# B&R Automation Studio project EFI (part 10)

#### AssignDataComms.st
```iecst
ACTION AssignDataComms:

	//Active modbus slave diagnosis when module ok (cable plugged). To set to false just unplug de cable
	IF PowerMeter.Status.Comms.xModuleOk THEN
		PowerMeter.Parameters.xActiveSlaveDiagnosis := TRUE; //1: Diagnosis enabled; 0=Reset diagnosis historic
	END_IF

	////////////////
	//Read Registers

	//Current
	IF PowerMeter.Status.Comms.xModuleOk THEN
		PowerMeter.Inputs.Comms.EffectiveCurrentPhaseA := PowerMeter.Inputs.Comms.ReceivedDataModPowerMeter[16];
		PowerMeter.Inputs.Comms.EffectiveCurrentPhaseB := PowerMeter.Inputs.Comms.ReceivedDataModPowerMeter[17];
		PowerMeter.Inputs.Comms.EffectiveCurrentPhaseC := PowerMeter.Inputs.Comms.ReceivedDataModPowerMeter[18];
		PowerMeter.Inputs.Comms.EffectiveCurrentNeutral := PowerMeter.Inputs.Comms.ReceivedDataModPowerMeter[19];
		PowerMeter.Inputs.Comms.MaxCurrentAllPhases := PowerMeter.Inputs.Comms.ReceivedDataModPowerMeter[20];
		PowerMeter.Inputs.Comms.IgEarthDefectiveCurrent := PowerMeter.Inputs.Comms.ReceivedDataModPowerMeter[21];
		PowerMeter.Inputs.Comms.CurrentDifferential := PowerMeter.Inputs.Comms.ReceivedDataModPowerMeter[22];
		PowerMeter.Inputs.Comms.MaxEffectiveCurrentPhaseA := PowerMeter.Inputs.Comms.ReceivedDataModPowerMeter[23];
		PowerMeter.Inputs.Comms.MaxEffectiveCurrentPhaseB := PowerMeter.Inputs.Comms.ReceivedDataModPowerMeter[24];
		PowerMeter.Inputs.Comms.MaxEffectiveCurrentPhaseC := PowerMeter.Inputs.Comms.ReceivedDataModPowerMeter[25];
		PowerMeter.Inputs.Comms.MaxEffectiveCurrentNeutral := PowerMeter.Inputs.Comms.ReceivedDataModPowerMeter[26];

		//Frequency
		PowerMeter.Inputs.Comms.MaxIgEarthDefectiveCurrent := PowerMeter.Inputs.Comms.ReceivedDataModPowerMeter[28];
		PowerMeter.Inputs.Comms.MaxCurrentDifferential := PowerMeter.Inputs.Comms.ReceivedDataModPowerMeter[29];

		//Voltage
		PowerMeter.Inputs.Comms.EffectiveVoltagePhasesAB := PowerMeter.Inputs.Comms.ReceivedDataModPowerMeter[30];
		PowerMeter.Inputs.Comms.EffectiveVoltagePhasesBC := PowerMeter.Inputs.Comms.ReceivedDataModPowerMeter[31];
		PowerMeter.Inputs.Comms.EffectiveVoltagePhasesCA := PowerMeter.Inputs.Comms.ReceivedDataModPowerMeter[32];
		PowerMeter.Inputs.Comms.EffectiveVoltagePhasesAN := PowerMeter.Inputs.Comms.ReceivedDataModPowerMeter[33];
		PowerMeter.Inputs.Comms.EffectiveVoltagePhasesBN := PowerMeter.Inputs.Comms.ReceivedDataModPowerMeter[34];
		PowerMeter.Inputs.Comms.EffectiveVoltagePhasesCN := PowerMeter.Inputs.Comms.ReceivedDataModPowerMeter[35];
		PowerMeter.Inputs.Comms.Frequency := PowerMeter.Inputs.Comms.ReceivedDataModPowerMeter[36]/10;
		PowerMeter.Inputs.Comms.FrequencyMax := PowerMeter.Inputs.Comms.ReceivedDataModPowerMeter[37]/10;

		//Power
		PowerMeter.Inputs.Comms.ActivePowerPhaseA := PowerMeter.Inputs.Comms.ReceivedDataModPowerMeter[38];
		PowerMeter.Inputs.Comms.ActivePowerPhaseB := PowerMeter.Inputs.Comms.ReceivedDataModPowerMeter[39];
		PowerMeter.Inputs.Comms.ActivePowerPhaseC := PowerMeter.Inputs.Comms.ReceivedDataModPowerMeter[40];
		PowerMeter.Inputs.Comms.TotalActivePower := PowerMeter.Inputs.Comms.ReceivedDataModPowerMeter[41];
		PowerMeter.Inputs.Comms.ApparentPowerPhaseA := PowerMeter.Inputs.Comms.ReceivedDataModPowerMeter[42];
		PowerMeter.Inputs.Comms.ApparentPowerPhaseB := PowerMeter.Inputs.Comms.ReceivedDataModPowerMeter[43];
		PowerMeter.Inputs.Comms.ApparentPowerPhaseC := PowerMeter.Inputs.Comms.ReceivedDataModPowerMeter[44];
		PowerMeter.Inputs.Comms.TotalApparentPower := PowerMeter.Inputs.Comms.ReceivedDataModPowerMeter[45];
		PowerMeter.Inputs.Comms.ReactivePowerPhaseA := PowerMeter.Inputs.Comms.ReceivedDataModPowerMeter[46];
		PowerMeter.Inputs.Comms.ReactivePowerPhaseB := PowerMeter.Inputs.Comms.ReceivedDataModPowerMeter[47];
		PowerMeter.Inputs.Comms.ReactivePowerPhaseC := PowerMeter.Inputs.Comms.ReceivedDataModPowerMeter[48];
		PowerMeter.Inputs.Comms.TotalReactivePower := PowerMeter.Inputs.Comms.ReceivedDataModPowerMeter[49];

		//Total Harmonic Distortion) (THD)
		PowerMeter.Inputs.Comms.THDVoltageAB := PowerMeter.Inputs.Comms.ReceivedDataModPowerMeter[104];
		PowerMeter.Inputs.Comms.THDVoltageBC := PowerMeter.Inputs.Comms.ReceivedDataModPowerMeter[105];
		PowerMeter.Inputs.Comms.THDVoltageCA := PowerMeter.Inputs.Comms.ReceivedDataModPowerMeter[106];
		PowerMeter.Inputs.Comms.THDVoltageAN := PowerMeter.Inputs.Comms.ReceivedDataModPowerMeter[107];
		PowerMeter.Inputs.Comms.THDVoltageBN := PowerMeter.Inputs.Comms.ReceivedDataModPowerMeter[108];
		PowerMeter.Inputs.Comms.THDVoltageCN := PowerMeter.Inputs.Comms.ReceivedDataModPowerMeter[109];
		PowerMeter.Inputs.Comms.THDCurrentA := PowerMeter.Inputs.Comms.ReceivedDataModPowerMeter[110];
		PowerMeter.Inputs.Comms.THDCurrentB := PowerMeter.Inputs.Comms.ReceivedDataModPowerMeter[111];
		PowerMeter.Inputs.Comms.THDCurrentC := PowerMeter.Inputs.Comms.ReceivedDataModPowerMeter[112];
		PowerMeter.Inputs.Comms.TotalTHDCurrent := PowerMeter.Inputs.Comms.ReceivedDataModPowerMeter[113];
	END_IF

END_ACTION
```

### Program Logical/ExtPack/_Extras/SafetyControllerCtrl/SafetyControllerCtrl_v1/SafetyControllerCtrl (IEC)

#### AssignDataComms.st
```iecst
ACTION AssignDataComms:

	//Active modbus slave diagnosis when module ok (cable plugged). To set to false just unplug de cable
	IF SafetyController.Status.Comms.xModuleOk THEN
		SafetyController.Parameters.xActiveSlaveDiagnosis := TRUE; //1: Diagnosis enabled; 0=Reset diagnosis historic
	END_IF

	//Pre bits treatment

	//Write Registers

	//Read Registers
	IF SafetyController.Status.Comms.xModuleOk THEN

		SafetyController.Inputs.Comms.FieldbusProbeStatus := DataFromSafety[11];

		IF NOT SafetyController.Parameters.xSimulationMode THEN
			//Software version
			SafetyController.Status.Version.0 := SafetyController.Inputs.Comms.FieldbusProbeStatus.0;
			SafetyController.Status.Version.1 := SafetyController.Inputs.Comms.FieldbusProbeStatus.1;
			SafetyController.Status.Version.2 := SafetyController.Inputs.Comms.FieldbusProbeStatus.2;
		END_IF

		CASE gMachine.Pt.ConfigNameID OF
			GC_CONFIG_1BK8BAR_NOZ2_ID:
				CASE SafetyController.Status.Version OF
					1: SafetyController.Status.Type := SAFETYCONTROLLERTY_DEFAULT;
					2: SafetyController.Status.Type := SAFETYCONTROLLERTY_DEFAULT;
					3: SafetyController.Status.Type := SAFETYCONTROLLERTY_CUBE_ALPHA;
					4: SafetyController.Status.Type := SAFETYCONTROLLERTY_SD;

					ELSE SafetyController.Status.Type := SAFETYCONTROLLERTY_UNDEFINED;
				END_CASE

			GC_CONFIG_1BK8BAR_NOZ2_AQ_ID:
				CASE SafetyController.Status.Version OF
					1: SafetyController.Status.Type := SAFETYCONTROLLERTY_NOZ2_AQ;

					ELSE SafetyController.Status.Type := SAFETYCONTROLLERTY_UNDEFINED;
				END_CASE

			GC_CONFIG_1BK7BAR_CUBE_ID:
				//To uncomment this code when first release that supports CUBE will be launched. So we will be sure safety controller version matches properly
				CASE SafetyController.Status.Version OF
					1: SafetyController.Status.Type := SAFETYCONTROLLERTY_CUBE;

					ELSE SafetyController.Status.Type := SAFETYCONTROLLERTY_UNDEFINED;
				END_CASE

			GC_CONFIG_1BK10BAR_MECANO_ID:
				//To uncomment this code when first release that supports CUBE will be launched. So we will be sure safety controller version matches properly
				CASE SafetyController.Status.Version OF
					1: SafetyController.Status.Type := SAFETYCONTROLLERTY_MECANO;

					ELSE SafetyController.Status.Type := SAFETYCONTROLLERTY_UNDEFINED;
				END_CASE

			GC_CONFIG_SIMTEST_ID:
				CASE gMachine.Pt.MachineModel OF
					Type_NOZ_2_AQ:
						SafetyController.Status.Type := SAFETYCONTROLLERTY_NOZ2_AQ;

					Type_NOZ_2_UV,
					Type_NOZ_2_UV_White:
						SafetyController.Status.Type := SAFETYCONTROLLERTY_DEFAULT;

					Type_CUBE,
					Type_CUBE_INSPECTION,
					Type_CUBE_GULLIVER,
					Type_CUBE_GULLIVER_INSPECTION:
						SafetyController.Status.Type := SAFETYCONTROLLERTY_CUBE;

					Type_MECANO_UV_WHITE,
					Type_MECANO_UV_OPV,
					Type_MECANO_UV_WHITE_OPV:
						SafetyController.Status.Type := SAFETYCONTROLLERTY_MECANO;

					ELSE SafetyController.Status.Type := SAFETYCONTROLLERTY_UNDEFINED;
				END_CASE

		END_CASE

		IF NOT SafetyController.Parameters.xSimulationMode THEN
			CASE SafetyController.Status.Type OF
				//Cube machine
				SAFETYCONTROLLERTY_CUBE:
					SafetyController.Inputs.Comms.SystemStatus := UINT_TO_USINT(DataFromSafety[0] AND 16#00FF);
					SafetyController.Inputs.Comms.ExpansionModule[0] := UINT_TO_USINT(DataFromSafety[1] AND 16#00FF); 			// CP0802
					SafetyController.Inputs.Comms.ExpansionModule[1] := UINT_TO_USINT(SHR((DataFromSafety[1] AND 16#FF00),8)); 	//DI16-0
					SafetyController.Inputs.Comms.ExpansionModule[2] := UINT_TO_USINT(DataFromSafety[2] AND 16#00FF);			//R04-0

					//Fieldbus probe
					//Inputs
					SafetyController.Inputs.xPrinterRearDoorSwitch := SafetyController.Inputs.Comms.FieldbusProbeStatus.3;
					SafetyController.Inputs.xPrinterMaintenanceKey := SafetyController.Inputs.Comms.FieldbusProbeStatus.4;
					SafetyController.Inputs.xHmiSwitch := SafetyController.Inputs.Comms.FieldbusProbeStatus.5;
					SafetyController.Inputs.xPrinterFrontDoorSwitch := SafetyController.Inputs.Comms.FieldbusProbeStatus.6;
					SafetyController.Inputs.xPrinterBacksideEstop := SafetyController.Inputs.Comms.FieldbusProbeStatus.7;
					SafetyController.Inputs.xPrinterFrontsideEstop := SafetyController.Inputs.Comms.FieldbusProbeStatus.8;
					SafetyController.Inputs.xX5Consent := SafetyController.Inputs.Comms.FieldbusProbeStatus.9;
					SafetyController.Inputs.xFanDoorSwitch := SafetyController.Inputs.Comms.FieldbusProbeStatus.12;

					//Outputs
					SafetyController.Outputs.xEnablePrinter1 := SafetyController.Inputs.Comms.FieldbusProbeStatus.11; //Revisar por qué esta asignación no funciona bien
					SafetyController.Outputs.xPrinterToX5 := SafetyController.Inputs.Comms.FieldbusProbeStatus.11;

				SAFETYCONTROLLERTY_DEFAULT,
				SAFETYCONTROLLERTY_CUBE_ALPHA,
				SAFETYCONTROLLERTY_SD:
					SafetyController.Inputs.Comms.SystemStatus := UINT_TO_USINT(DataFromSafety[0] AND 16#00FF);
					SafetyController.Inputs.Comms.ExpansionModule[0] := UINT_TO_USINT(DataFromSafety[1] AND 16#00FF);			// CP0802
					SafetyController.Inputs.Comms.ExpansionModule[1] := UINT_TO_USINT(SHR((DataFromSafety[1] AND 16#FF00),8));	//MX0802
					SafetyController.Inputs.Comms.ExpansionModule[2] := UINT_TO_USINT(DataFromSafety[2] AND 16#00FF);			//DI16-0
					SafetyController.Inputs.Comms.ExpansionModule[3] := UINT_TO_USINT(SHR((DataFromSafety[2] AND 16#FF00),8));	//DI16-1
					SafetyController.Inputs.Comms.ExpansionModule[4] := UINT_TO_USINT(DataFromSafety[3] AND 16#00FF);			//R04-0
					SafetyController.Inputs.Comms.ExpansionModule[5] := UINT_TO_USINT(SHR((DataFromSafety[3] AND 16#FF00),8));	//R04-1
					SafetyController.Inputs.Comms.ExpansionModule[6] := UINT_TO_USINT(DataFromSafety[4] AND 16#00FF);			//R04-2

					//SafetyController.Inputs.Comms.FieldbusProbeStatus := DataFromSafety[11];
					SafetyController.Inputs.Comms.OSSDStatus := DataFromSafety[13];
					SafetyController.Inputs.Comms.DiagnosticCode := DataFromSafety[14];

					//Post bit treatment
					//Fieldbus: Currently there is no need to acknowledge fiedlbus inputs set in SoSafe program so info coming from inputs is enough

					//Modules physical inputs
					//Ancillaries
					SafetyController.Inputs.xFeederEstop			:= SafetyController.Inputs.Comms.FieldbusProbeStatus.8; //SafetyController.Inputs.Comms.ExpansionModule[1].0;
					SafetyController.Inputs.xPrimerEstop 			:= SafetyController.Inputs.Comms.FieldbusProbeStatus.9; //SafetyController.Inputs.Comms.ExpansionModule[1].2;
					SafetyController.Inputs.xOvervarnishEstop 		:= SafetyController.Inputs.Comms.FieldbusProbeStatus.14; //SafetyController.Inputs.Comms.ExpansionModule[2].4;
					SafetyController.Inputs.xStackerEstop 			:= SafetyController.Inputs.Comms.FieldbusProbeStatus.15; //SafetyController.Inputs.Comms.ExpansionModule[2].0;
					SafetyController.Inputs.xSarmEstop				:= SafetyController.Inputs.Comms.FieldbusProbeStatus.7;

					//Dryer
					SafetyController.Inputs.xDryerBacksideEstop 	:= SafetyController.Inputs.Comms.FieldbusProbeStatus.12; //SafetyController.Inputs.Comms.ExpansionModule[1].4;
					SafetyController.Inputs.xDryerFrontsideEstop 	:= SafetyController.Inputs.Comms.FieldbusProbeStatus.13; //SafetyController.Inputs.Comms.ExpansionModule[1].6;
					SafetyController.Inputs.xDryerFrontDoorSwitch1	:= SafetyController.Inputs.Comms.FieldbusProbeStatus.3; //SafetyController.Inputs.Comms.ExpansionModule[2].6;
					SafetyController.Inputs.xDryerFrontDoorSwitch2	:= SafetyController.Inputs.Comms.FieldbusProbeStatus.4; //SafetyController.Inputs.Comms.ExpansionModule[3].4;
					SafetyController.Inputs.xDryerBackDoorSwitch1	:= SafetyController.Inputs.Comms.FieldbusProbeStatus.5; //SafetyController.Inputs.Comms.ExpansionModule[3].6;
					SafetyController.Inputs.xDryerBackDoorSwitch2	:= SafetyController.Inputs.Comms.FieldbusProbeStatus.6; //SafetyController.Inputs.Comms.ExpansionModule[4].0;
					SafetyController.Inputs.xDryerMaintenanceKey	:= SafetyController.Inputs.Comms.ExpansionModule[4].3;
					SafetyController.Inputs.xDryerBlowersEnable		:= SafetyController.Inputs.Comms.ExpansionModule[2].3;

					//Printer
					SafetyController.Inputs.xPrinterMaintenanceKey 	:= SafetyController.Inputs.Comms.ExpansionModule[4].2;
					SafetyController.Inputs.xPrinterBlowersEnable	:= SafetyController.Inputs.Comms.ExpansionModule[2].2;
					SafetyController.Inputs.xPrinterBlowersSwitch	:= TRUE; //SafetyController.Inputs.Comms.FieldbusProbeStatus.2;
					SafetyController.Inputs.xPrinterLightCurtain 	:= SafetyController.Inputs.Comms.ExpansionModule[0].0;
					SafetyController.Inputs.xPrinterDoorLock 		:= SafetyController.Inputs.Comms.ExpansionModule[0].2;
					SafetyController.Inputs.xPrinterBacksideEstop 	:= SafetyController.Inputs.Comms.FieldbusProbeStatus.10;
					SafetyController.Inputs.xPrinterFrontsideEstop 	:= SafetyController.Inputs.Comms.FieldbusProbeStatus.11;

					//OSSD Outputs
					SafetyController.Outputs.xEnablePrinter1 := SafetyController.Inputs.Comms.OSSDStatus.0;
					//SafetyController.Outputs.xEnablePrinter2 := SafetyController.Inputs.Comms.OSSDStatus.1;
					SafetyController.Outputs.xEnablePrinterBlowers1 := SafetyController.Inputs.Comms.OSSDStatus.1;
					//SafetyController.Outputs.xEnablePrinterBlowers2	:= SafetyController.Inputs.Comms.OSSDStatus.3;
					SafetyController.Outputs.xEnableDryer1	:= SafetyController.Inputs.Comms.OSSDStatus.2;
					//SafetyController.Outputs.xEnableDryer2	:= SafetyController.Inputs.Comms.OSSDStatus.5;

				SAFETYCONTROLLERTY_MECANO:
					SafetyController.Inputs.Comms.SystemStatus := UINT_TO_USINT(DataFromSafety[0] AND 16#00FF);
					SafetyController.Inputs.Comms.ExpansionModule[0] := UINT_TO_USINT(DataFromSafety[1] AND 16#00FF);			// CP0802
					SafetyController.Inputs.Comms.ExpansionModule[1] := UINT_TO_USINT(SHR((DataFromSafety[1] AND 16#FF00),8));	//MX0802
					SafetyController.Inputs.Comms.ExpansionModule[2] := UINT_TO_USINT(DataFromSafety[2] AND 16#00FF);			//DI16-0
					SafetyController.Inputs.Comms.ExpansionModule[3] := UINT_TO_USINT(SHR((DataFromSafety[2] AND 16#FF00),8));	//DI16-1
					SafetyController.Inputs.Comms.ExpansionModule[4] := UINT_TO_USINT(DataFromSafety[3] AND 16#00FF);			//R04-0
					SafetyController.Inputs.Comms.ExpansionModule[5] := UINT_TO_USINT(SHR((DataFromSafety[3] AND 16#FF00),8));	//R04-1
					SafetyController.Inputs.Comms.ExpansionModule[6] := UINT_TO_USINT(DataFromSafety[4] AND 16#00FF);			//R04-2

					//SafetyController.Inputs.Comms.FieldbusProbeStatus := DataFromSafety[11];
					SafetyController.Inputs.Comms.OSSDStatus := DataFromSafety[13];
					SafetyController.Inputs.Comms.DiagnosticCode := DataFromSafety[14];

					//Post bit treatment
					//Modules physical inputs
					//Ancillaries
					SafetyController.Inputs.xFeederEstop			:= SafetyController.Inputs.Comms.FieldbusProbeStatus.8;
					SafetyController.Inputs.xPrimerEstop 			:= SafetyController.Inputs.Comms.FieldbusProbeStatus.9;
					SafetyController.Inputs.xOvervarnishEstop 		:= SafetyController.Inputs.Comms.FieldbusProbeStatus.14;
					SafetyController.Inputs.xStackerEstop 			:= SafetyController.Inputs.Comms.FieldbusProbeStatus.15;
					SafetyController.Inputs.xSarmEstop				:= SafetyController.Inputs.Comms.FieldbusProbeStatus.7;

					//Printer
					SafetyController.Inputs.xPrinterMaintenanceKey 	:= SafetyController.Inputs.Comms.FieldbusProbeStatus.5;
					SafetyController.Inputs.xPrinterBlowersEnable	:= SafetyController.Inputs.Comms.ExpansionModule[2].2;
					SafetyController.Inputs.xPrinterBlowersSwitch	:= SafetyController.Inputs.Comms.FieldbusProbeStatus.6;
					SafetyController.Inputs.xPrinterLightCurtain 	:= SafetyController.Inputs.Comms.FieldbusProbeStatus.3;
					SafetyController.Inputs.xPrinterDoorLock 		:= SafetyController.Inputs.Comms.FieldbusProbeStatus.4;
					SafetyController.Inputs.xPrinterBacksideEstop 	:= SafetyController.Inputs.Comms.FieldbusProbeStatus.10;
					SafetyController.Inputs.xPrinterFrontsideEstop 	:= SafetyController.Inputs.Comms.FieldbusProbeStatus.11;

					//OSSD Outputs
					SafetyController.Outputs.xEnablePrinter1 		:= SafetyController.Inputs.Comms.OSSDStatus.0;
					SafetyController.Outputs.xEnablePrinterBlowers1 := SafetyController.Inputs.Comms.OSSDStatus.1;

				SAFETYCONTROLLERTY_NOZ2_AQ:
					SafetyController.Inputs.Comms.SystemStatus := UINT_TO_USINT(DataFromSafety[0] AND 16#00FF);
					SafetyController.Inputs.Comms.ExpansionModule[0] := UINT_TO_USINT(DataFromSafety[1] AND 16#00FF);			// CP0802
					SafetyController.Inputs.Comms.ExpansionModule[1] := UINT_TO_USINT(SHR((DataFromSafety[1] AND 16#FF00),8));	//MX0802
					SafetyController.Inputs.Comms.ExpansionModule[2] := UINT_TO_USINT(DataFromSafety[2] AND 16#00FF);			//DI16-0
					SafetyController.Inputs.Comms.ExpansionModule[3] := UINT_TO_USINT(SHR((DataFromSafety[2] AND 16#FF00),8));	//DI16-1
					SafetyController.Inputs.Comms.ExpansionModule[4] := UINT_TO_USINT(DataFromSafety[3] AND 16#00FF);			//R04-0
					SafetyController.Inputs.Comms.ExpansionModule[5] := UINT_TO_USINT(SHR((DataFromSafety[3] AND 16#FF00),8));	//R04-1
					SafetyController.Inputs.Comms.ExpansionModule[6] := UINT_TO_USINT(DataFromSafety[4] AND 16#00FF);			//R04-2

					SafetyController.Inputs.Comms.OSSDStatus := DataFromSafety[13];
					SafetyController.Inputs.Comms.DiagnosticCode := DataFromSafety[14];

					//Post bit treatment
					//Fieldbus: Currently there is no need to acknowledge fiedlbus inputs set in SoSafe program so info coming from inputs is enough

					//Modules physical inputs
					//Ancillaries
					SafetyController.Inputs.xFeederEstop			:= SafetyController.Inputs.Comms.FieldbusProbeStatus.8; //SafetyController.Inputs.Comms.ExpansionModule[1].0;
					SafetyController.Inputs.xPrimerEstop 			:= SafetyController.Inputs.Comms.FieldbusProbeStatus.9; //SafetyController.Inputs.Comms.ExpansionModule[1].2;
					SafetyController.Inputs.xOvervarnishEstop 		:= SafetyController.Inputs.Comms.FieldbusProbeStatus.14; //SafetyController.Inputs.Comms.ExpansionModule[2].4;
					SafetyController.Inputs.xStackerEstop 			:= SafetyController.Inputs.Comms.FieldbusProbeStatus.15; //SafetyController.Inputs.Comms.ExpansionModule[2].0;

					//Dryer
					SafetyController.Inputs.xDryerBacksideEstop 	:= SafetyController.Inputs.Comms.FieldbusProbeStatus.12; //SafetyController.Inputs.Comms.ExpansionModule[1].4;
					SafetyController.Inputs.xDryerFrontsideEstop 	:= SafetyController.Inputs.Comms.FieldbusProbeStatus.13; //SafetyController.Inputs.Comms.ExpansionModule[1].6;
					SafetyController.Inputs.xDryerFrontDoorSwitch1	:= SafetyController.Inputs.Comms.FieldbusProbeStatus.3; //SafetyController.Inputs.Comms.ExpansionModule[2].6;
					SafetyController.Inputs.xDryerFrontDoorSwitch2	:= SafetyController.Inputs.Comms.FieldbusProbeStatus.4; //SafetyController.Inputs.Comms.ExpansionModule[3].4;
					SafetyController.Inputs.xDryerBackDoorSwitch1	:= SafetyController.Inputs.Comms.FieldbusProbeStatus.5; //SafetyController.Inputs.Comms.ExpansionModule[3].6;
					SafetyController.Inputs.xDryerBackDoorSwitch2	:= SafetyController.Inputs.Comms.FieldbusProbeStatus.6; //SafetyController.Inputs.Comms.ExpansionModule[4].0;
					SafetyController.Inputs.xDryerMaintenanceKey	:= SafetyController.Inputs.Comms.ExpansionModule[4].3;
					SafetyController.Inputs.xDryerBlowersEnable		:= SafetyController.Inputs.Comms.ExpansionModule[2].3;

					//Printer
					SafetyController.Inputs.xPrinterMaintenanceKey 	:= SafetyController.Inputs.Comms.ExpansionModule[4].2;
					SafetyController.Inputs.xPrinterBlowersEnable	:= SafetyController.Inputs.Comms.ExpansionModule[2].2;
					SafetyController.Inputs.xPrinterBlowersSwitch	:= TRUE;
					SafetyController.Inputs.xPrinterLightCurtain 	:= SafetyController.Inputs.Comms.ExpansionModule[0].0;
					SafetyController.Inputs.xPrinterDoorLock 		:= SafetyController.Inputs.Comms.ExpansionModule[0].2;
					SafetyController.Inputs.xPrinterBacksideEstop 	:= SafetyController.Inputs.Comms.FieldbusProbeStatus.10;
					SafetyController.Inputs.xPrinterFrontsideEstop 	:= SafetyController.Inputs.Comms.FieldbusProbeStatus.11;

					//OSSD Outputs
					SafetyController.Outputs.xEnablePrinter1 := SafetyController.Inputs.Comms.OSSDStatus.0;
					SafetyController.Outputs.xEnablePrinterBlowers1 := SafetyController.Inputs.Comms.OSSDStatus.1;
					SafetyController.Outputs.xEnableDryer1	:= SafetyController.Inputs.Comms.OSSDStatus.2;

				ELSE
					SafetyController.Inputs := ResetSafetyInputs;
					SafetyController.Outputs := ResetSafetyOutputs;

			END_CASE
		END_IF
	END_IF

END_ACTION
```

#### Alarms.st
```iecst
ACTION Alarms:

	//Reset Alarms with an external order to reset
	IF SafetyController.Commands.xReset THEN
		ResetAlarms;
	END_IF

	//Saving modbus slave status when comms error raises
	IF EDGEPOS (SafetyController.Alarms.xCommsError) THEN
		ModSlaveState := SafetyController.Status.Comms.ModSlaveState;
		LastError := SafetyController.Status.Comms.LastError;
		LastErrorBlockNum := SafetyController.Status.Comms.LastErrorBlockNum;
	END_IF

	//Alarms related to comms
	IF SafetyController.Status.Comms.xModuleOk THEN

		CASE SafetyController.Status.Type OF
			//Cube machine
			SAFETYCONTROLLERTY_CUBE:

				SafetyController.Alarms.xAlrPrinterRearDoorSwitch := NOT SafetyController.Inputs.xPrinterRearDoorSwitch AND NOT SafetyController.Inputs.xPrinterMaintenanceKey;
				SafetyController.Alarms.xAlrHmiSwitch := NOT SafetyController.Inputs.xHmiSwitch;
				SafetyController.Alarms.xAlrPrinterFrontDoorSwitch := NOT SafetyController.Inputs.xPrinterFrontDoorSwitch AND NOT SafetyController.Inputs.xPrinterMaintenanceKey;
				SafetyController.Alarms.xAlrPrinterFanDoorSwitch := NOT SafetyController.Inputs.xFanDoorSwitch;

				SafetyController.Alarms.xAlrPrinterEStops := 	NOT SafetyController.Inputs.xPrinterBacksideEstop OR
																NOT SafetyController.Inputs.xPrinterFrontsideEstop;

				SafetyController.Alarms.xAlrPrinter := 	SafetyController.Alarms.xAlrPrinterRearDoorSwitch OR
														SafetyController.Alarms.xAlrHmiSwitch OR
														SafetyController.Alarms.xAlrPrinterFrontDoorSwitch OR
														SafetyController.Alarms.xAlrPrinterFanDoorSwitch OR
														SafetyController.Alarms.xAlrPrinterEStops;

				SafetyController.Alarms.xAlrPrinterDoorLockKeyActivated := SafetyController.Inputs.xPrinterMaintenanceKey;

				SafetyController.Alarms.xAlrFeeder := NOT SafetyController.Inputs.xX5Consent;

				SafetyController.Alarms.xAlrPrinterFrontEstop :=  NOT SafetyController.Inputs.xPrinterFrontsideEstop;
				SafetyController.Alarms.xAlrPrinterRearEstop := NOT SafetyController.Inputs.xPrinterBacksideEstop;

			SAFETYCONTROLLERTY_DEFAULT,
			SAFETYCONTROLLERTY_CUBE_ALPHA,
			SAFETYCONTROLLERTY_SD,
			SAFETYCONTROLLERTY_MECANO:
				tonAlarmFeeder.IN := NOT SafetyController.Inputs.xFeederEstop;
				tonAlarmFeeder.PT := T#3s;
				tonAlarmFeeder();
				SafetyController.Alarms.xAlrFeeder := tonAlarmFeeder.Q;

				tonAlarmPrimer.IN := NOT SafetyController.Inputs.xPrimerEstop;
				tonAlarmPrimer.PT := T#3s;
				tonAlarmPrimer();
				SafetyController.Alarms.xAlrPrimer := tonAlarmPrimer.Q;

				SafetyController.Alarms.xAlrPrinter := 	NOT SafetyController.Inputs.xPrinterLightCurtain OR
														NOT SafetyController.Inputs.xPrinterDoorLock OR
														NOT SafetyController.Inputs.xPrinterBacksideEstop OR
														NOT SafetyController.Inputs.xPrinterFrontsideEstop;

				SafetyController.Alarms.xAlrPrinterEStops := 	NOT SafetyController.Inputs.xPrinterBacksideEstop OR
																NOT SafetyController.Inputs.xPrinterFrontsideEstop;

				tonAlarmOverVarnish.IN := NOT SafetyController.Inputs.xOvervarnishEstop;
				tonAlarmOverVarnish.PT := T#3s;
				tonAlarmOverVarnish();
				SafetyController.Alarms.xAlrOverVarnish := tonAlarmOverVarnish.Q;

				tonAlarmStacker.IN := NOT SafetyController.Inputs.xStackerEstop;
				tonAlarmStacker.PT := T#3s;
				tonAlarmStacker();
				SafetyController.Alarms.xAlrStacker := tonAlarmStacker.Q;

				IF SafetyController.Status.Type = SAFETYCONTROLLERTY_SD OR SafetyController.Status.Type = SAFETYCONTROLLERTY_MECANO THEN
					tonAlarmSarm.IN := NOT SafetyController.Inputs.xSarmEstop;
					tonAlarmSarm.PT := T#3s;
					tonAlarmSarm();
					SafetyController.Alarms.xAlrSarm := tonAlarmSarm.Q;
				END_IF

				IF NOT gMachine.St.Mode.xZero THEN
					SafetyController.Alarms.xAlrPrinterDoorLock := NOT SafetyController.Inputs.xPrinterDoorLock;
					//SafetyController.Alarms.xAlrPrinterLightCurtain := NOT SafetyController.Inputs.xPrinterLightCurtain;
				END_IF

				SafetyController.Alarms.xAlrPrinterDoorLockKeyActivated := SafetyController.Inputs.xPrinterMaintenanceKey;
				IF SafetyController.Status.Type <> SAFETYCONTROLLERTY_CUBE_ALPHA THEN
					SafetyController.Alarms.xAlrBlowersEnclosureSwitchOff := NOT SafetyController.Inputs.xPrinterBlowersSwitch;
				END_IF

			SAFETYCONTROLLERTY_NOZ2_AQ:
				tonAlarmFeeder.IN := NOT SafetyController.Inputs.xFeederEstop;
				tonAlarmFeeder.PT := T#3s;
				tonAlarmFeeder();
				SafetyController.Alarms.xAlrFeeder := tonAlarmFeeder.Q;

				tonAlarmPrimer.IN := NOT SafetyController.Inputs.xPrimerEstop;
				tonAlarmPrimer.PT := T#3s;
				tonAlarmPrimer();
				SafetyController.Alarms.xAlrPrimer := tonAlarmPrimer.Q;

				SafetyController.Alarms.xAlrPrinter := 	NOT SafetyController.Inputs.xPrinterLightCurtain OR
														NOT SafetyController.Inputs.xPrinterDoorLock OR
														NOT SafetyController.Inputs.xPrinterBacksideEstop OR
														NOT SafetyController.Inputs.xPrinterFrontsideEstop;

				SafetyController.Alarms.xAlrPrinterEStops := 	NOT SafetyController.Inputs.xPrinterBacksideEstop OR
																NOT SafetyController.Inputs.xPrinterFrontsideEstop;

				tonAlarmDryer.IN := NOT SafetyController.Inputs.xDryerBacksideEstop OR NOT SafetyController.Inputs.xDryerFrontsideEstop;
				tonAlarmDryer.PT := T#3s;
				tonAlarmDryer();
				SafetyController.Alarms.xAlrDryer := tonAlarmDryer.Q;

				tonAlarmOverVarnish.IN := NOT SafetyController.Inputs.xOvervarnishEstop;
				tonAlarmOverVarnish.PT := T#3s;
				tonAlarmOverVarnish();
				SafetyController.Alarms.xAlrOverVarnish := tonAlarmOverVarnish.Q;

				tonAlarmStacker.IN := NOT SafetyController.Inputs.xStackerEstop;
				tonAlarmStacker.PT := T#3s;
				tonAlarmStacker();
				SafetyController.Alarms.xAlrStacker := tonAlarmStacker.Q;

				IF NOT gMachine.St.Mode.xZero THEN
					SafetyController.Alarms.xAlrPrinterDoorLock := NOT SafetyController.Inputs.xPrinterDoorLock;
					//SafetyController.Alarms.xAlrPrinterLightCurtain := NOT SafetyController.Inputs.xPrinterLightCurtain;
				END_IF

				SafetyController.Alarms.xAlrPrinterDoorLockKeyActivated := SafetyController.Inputs.xPrinterMaintenanceKey;
				SafetyController.Alarms.xAlrBlowersEnclosureSwitchOff := NOT SafetyController.Inputs.xPrinterBlowersSwitch;

		END_CASE
	END_IF

	//Alarm related to comms
	ton_CommsError.IN := NOT SafetyController.Orders.xDisableReadBlock AND NOT SafetyController.Status.Comms.xModuleOk;
	ton_CommsError.PT := T#200ms;
	ton_CommsError();
	IF ton_CommsError.Q THEN SafetyController.Alarms.xCommsError := TRUE; END_IF

	iReasonCritical.0 := SafetyController.Alarms.xAlrFeeder;
	iReasonCritical.1 := SafetyController.Alarms.xAlrPrimer;
	iReasonCritical.2 := SafetyController.Alarms.xAlrPrinter;
	iReasonCritical.3 := SafetyController.Alarms.xAlrDryer;
	iReasonCritical.4 := SafetyController.Alarms.xAlrOverVarnish;
	iReasonCritical.5 := SafetyController.Alarms.xAlrStacker;
	iReasonCritical.6 := SafetyController.Alarms.xCommsError;

	IF iReasonCritical>0 THEN
		SafetyController.Alarms.xCriticalAlarm := TRUE ;
	END_IF

END_ACTION

ACTION ResetAlarms:
	SafetyController.Alarms := AlarmsReseted;
END_ACTION
```

#### SafetyController.var - Local variables
```iecst
VAR
	SafetyController : REFERENCE TO stSafetyController;
	DataFromSafety : REFERENCE TO ARRAY[0..20] OF UINT;
	CommsReset : SafetyControllerCommsInputs_typ;
	ModSlaveState : UINT;
	LastError : UINT;
	LastErrorBlockNum : UINT;
	AlarmsReseted : SafetyControllerAlarms_typ;
	tonAlarmFeeder : TON;
	tonAlarmPrimer : TON;
	tonAlarmOverVarnish : TON;
	tonAlarmDryer : TON;
	tonAlarmStacker : TON;
	tonAlarmSarm : TON;
	iReasonCritical : UINT;
	ton_CommsError : TON;
	ResetSafetyOutputs : SafetyControllerOutputs_typ;
	ResetSafetyInputs : SafetyControllerInputs_typ;
END_VAR
```

### SafetyControllerSim.typ
```iecst
TYPE
	SafetyControllerSim_typ : 	STRUCT
		Commands : SafetyControllerSimCommands_typ;
		Inputs : SafetyControllerInputs_typ;
		Outputs : SafetyControllerOutputs_typ;
	END_STRUCT;
	SafetyControllerSimCommands_typ : 	STRUCT
		xSafetyToDefault : BOOL; (*To set in simulation all the inputs to have the Safety OK*)
	END_STRUCT;
	SafetyControllerSimOutputs_typ : 	STRUCT
		xEnablePrinter1 : BOOL; (*OSSD*)
		xEnablePrinter2 : BOOL; (*OSSD*)
		xEnablePrinterBlowers1 : BOOL; (*OSSD*)
		xEnablePrinterBlowers2 : BOOL; (*OSSD*)
		xEnableDryer1 : BOOL; (*OSSD*)
		xEnableDryer2 : BOOL; (*OSSD*)
		xEnableDryerBlowers1 : BOOL; (*OSSD*)
		xEnableDryerBlowers2 : BOOL; (*OSSD*)
		xFeederToLine1 : BOOL; (*Relay*)
		xFeederToLine2 : BOOL; (*Relay*)
		xLineToFeeder1 : BOOL; (*Relay*)
		xLineToFeeder2 : BOOL; (*Relay*)
		xPrimerToLine1 : BOOL; (*Relay*)
		xPrimerToLine2 : BOOL; (*Relay*)
		xLineToPrimer1 : BOOL; (*Relay*)
		xLineToPrimer2 : BOOL; (*Relay*)
		xStackerToLine1 : BOOL; (*Relay*)
		xStackerToLine2 : BOOL; (*Relay*)
		xLineToStacker1 : BOOL; (*Relay*)
		xLineToStacker2 : BOOL; (*Relay*)
		xIRToLine1 : BOOL; (*Relay*)
		xIRToLine2 : BOOL; (*Relay*)
		xLineToIR1 : BOOL; (*Relay*)
		xLineToIR2 : BOOL; (*Relay*)
		xUVToLine1 : BOOL; (*Relay*)
		xUVToLine2 : BOOL; (*Relay*)
		xLineToUV1 : BOOL; (*Relay*)
		xLineToUV2 : BOOL; (*Relay*)
		xPrinterToX5 : BOOL; (*Relay*)
	END_STRUCT;
END_TYPE
```

### Program Logical/ExtPack/_Extras/SafetyControllerCtrl/SafetyControllerSim/SafetyControllerSim_v1/SafetyControllerSim (IEC)

#### SafetyControllerSim.var - Local variables
```iecst
VAR
	SimSafetyController : REFERENCE TO SafetyControllerSim_typ;
	SafetyController : REFERENCE TO stSafetyController;
	DataFromSimSafety : REFERENCE TO ARRAY[0..20] OF UINT;
END_VAR
```

### Program Logical/ExtPack/_Media/ThicknessCtrl/ThickLib

#### ThicknessCtrlConstants.var
```iecst
VAR CONSTANT
	THICK_MEDIATRACKING_MAX_MEDIA : USINT := 20; (*Maximum quantity of different media inside the machine. This value could be critical with really small media and long machines*)
	THICK_MEDIATRACKING_MAX_MEDIA_x2 : USINT := 2*THICK_MEDIATRACKING_MAX_MEDIA; (*Maximum quantity of different media inside the machine. This value could be critical with really small media and long machines*)
	THICK_MAX_UPDATE_VALUES : USINT := 10; (*Maximum quantity of the updated values to be managed by the machine due to max speed and scan cycle*)
	THICK_MAX_TRACKING_EVENTS : USINT := 20; (*Maximum quantity of the EVENTS*)
	INDEXCURING_L1_COLOR : USINT := 0; (*Matrix with the information about media that need to be cured. Each position corresponds to a cm. Bit 0: L1 Color, Bit 1 L1 White, Bit 2 L1 Primer, Bit 3 L2 Color, Bit 4 L2 White, Bit 5 L2 Primer*)
	INDEXCURING_L1_WHITE : USINT := 1; (*Matrix with the information about media that need to be cured. Each position corresponds to a cm. Bit 0: L1 Color, Bit 1 L1 White, Bit 2 L1 Primer, Bit 3 L2 Color, Bit 4 L2 White, Bit 5 L2 Primer*)
	INDEXCURING_L1_PRIMER : USINT := 2; (*Matrix with the information about media that need to be cured. Each position corresponds to a cm. Bit 0: L1 Color, Bit 1 L1 White, Bit 2 L1 Primer, Bit 3 L2 Color, Bit 4 L2 White, Bit 5 L2 Primer*)
	INDEXCURING_L2_COLOR : USINT := 3; (*Matrix with the information about media that need to be cured. Each position corresponds to a cm. Bit 0: L1 Color, Bit 1 L1 White, Bit 2 L1 Primer, Bit 3 L2 Color, Bit 4 L2 White, Bit 5 L2 Primer*)
	INDEXCURING_L2_WHITE : USINT := 4; (*Matrix with the information about media that need to be cured. Each position corresponds to a cm. Bit 0: L1 Color, Bit 1 L1 White, Bit 2 L1 Primer, Bit 3 L2 Color, Bit 4 L2 White, Bit 5 L2 Primer*)
	INDEXCURING_L2_PRIMER : USINT := 5; (*Matrix with the information about media that need to be cured. Each position corresponds to a cm. Bit 0: L1 Color, Bit 1 L1 White, Bit 2 L1 Primer, Bit 3 L2 Color, Bit 4 L2 White, Bit 5 L2 Primer*)
	INDEXTRACKING_L1 : USINT := 0; (*Matrix with the information about media tracking. Each position corresponds to a cm. Bit 0: L1 , Bit 1 L2*)
	INDEXTRACKING_L2 : USINT := 1; (*Matrix with the information about media tracking. Each position corresponds to a cm. Bit 0: L1 , Bit 1 L2*)
	THICKENERGY_MAX_CROSS : USINT := 140; (*With a discretization of 10mm, with 140 elements we cover 1400mm*)
	THICKENERGY_MAX_CROSS_ITEMS : USINT := THICKENERGY_MAX_CROSS-1; (*In an array stating in 0, the last element is 1 less than the quantity of elements*)
	THICKENERGY_MAX_PROCESS : USINT := 70; (*With a discretization of 50mm, with 70 elements we achive 3500mm*)
	THICKENERGY_MAX_PROCESS_ITEMS : USINT := THICKENERGY_MAX_PROCESS-1; (*In an array stating in 0, the last element is 1 less than the quantity of elements*)
	THICKENERGY_CROSS_STEP : USINT := 10; (*Value in mm*)
	THICKENERGY_PROCESS_STEP : USINT := 5; (*Value in cm*)
	THICKENERGY_MAX_LAMPS : USINT := 65; (*Max NIR lamps in all configurations. Lamp 1 is the one closer to operator*)
END_VAR
```

#### AssignStack.st
```iecst
FUNCTION AssignItemInStack

	AssignItemInStack := AssignItemEnergyInStack(ADR(ItemMedia), ADR(ItemEnergyFake), ADR(StackArray), 0, Position, 0);

END_FUNCTION

FUNCTION AssignItemEnergyInStack

	// Manage Energy information
	IF ADR(EnergyArray) > 0 THEN
		EnergyArray[PositionEnergy] := ItemEnergy;
		StackArray[PositionStack].iIndexMediaEnergy := PositionEnergy;
		StackArray[PositionStack].pMediaEnery := ADR(EnergyArray[PositionEnergy]);
	ELSE
		StackArray[PositionStack].iIndexMediaEnergy := 0;
		StackArray[PositionStack].pMediaEnery := 0;
	END_IF

	// Manage Media information
	StackArray[PositionStack].Media := ItemMedia;

	AssignItemEnergyInStack := 0;

END_FUNCTION

FUNCTION AssignLastItemInStack

	AssignLastItemInStack := AssignLastItemEnergyInStack(ADR(ItemMedia), ADR(ItemEnergyFake), ADR(StackArray), 0, TotalElementsStack, IndexEnergyFake);

END_FUNCTION

FUNCTION AssignLastItemEnergyInStack

	// Check if the item NOT inside the array
	AssignLastItemEnergyInStack := CheckNotItemInStack(ItemMedia.id, ADR(StackArray), TotalElementsStack, PositionFound);
	IF AssignLastItemEnergyInStack <> 0 THEN
		RETURN;
	END_IF

	AssignLastItemEnergyInStack := AssignItemEnergyInStack(ADR(ItemMedia), ADR(ItemEnergy), ADR(StackArray), ADR(EnergyArray), TotalElementsStack, IndexEnergy);

	// Manage Energy index
	IF ADR(EnergyArray) > 0 THEN
		IndexEnergy := IndexEnergy + 1;
		IF IndexEnergy > THICK_MEDIATRACKING_MAX_MEDIA_x2 THEN
			IndexEnergy := 0;
		END_IF
	END_IF

	// Manage Stack index
	TotalElementsStack := TotalElementsStack + 1;

END_FUNCTION

FUNCTION InsertItemInStack

	InsertItemInStack := InsertItemEnergyInStack(Id, ADR(ItemMedia), ADR(ItemEnergyFake), ADR(StackArray), 0, TotalElementsStack, IndexEnergyFake);

END_FUNCTION

FUNCTION InsertItemEnergyInStack

	// Check if the item inside the array
	CheckResult := CheckItemInStack(Id, ADR(StackArray), TotalElementsStack, PositionFound);
	IF CheckResult <> 0 THEN
		InsertItemEnergyInStack := CheckResult;
		RETURN;
	END_IF

	// Check if the item NOT inside the array
	CheckResult := CheckNotItemInStack(ItemMedia.id, ADR(StackArray), TotalElementsStack, PositionFound);
	IF CheckResult <> 0 THEN
		InsertItemEnergyInStack := CheckResult;
		RETURN;
	END_IF

	//Make space in Stack
	ShiftArrayOffset(ADR(StackArray), SIZEOF(StackArray), SIZEOF(StackArray[0]), PositionFound+1, PositionFound+2, TotalElementsStack - PositionFound -1);

	//Assing information
	AssignItemEnergyInStack(ADR(ItemMedia), ADR(ItemEnergy), ADR(StackArray), ADR(EnergyArray), PositionFound+1, IndexEnergy);

	// Manage Energy index
	IF ADR(EnergyArray) > 0 THEN
		IndexEnergy := IndexEnergy + 1;
		IF IndexEnergy > THICK_MEDIATRACKING_MAX_MEDIA_x2 THEN
			IndexEnergy := 0;
		END_IF
	END_IF

	// Manage Stack index
	TotalElementsStack := TotalElementsStack + 1;

	InsertItemEnergyInStack := 0;

END_FUNCTION

FUNCTION RemoveItemInStack

	// Directly remove everything if asked
	IF Id = -1 THEN
		// Clean all the array
		brsmemset(ADR(StackArray), 0, SIZEOF(StackArray));
		TotalElementsStack := 0;
		RemoveItemInStack := 0;
		RETURN;
	END_IF

	// Check if the item inside the array
	CheckResult := CheckItemInStack(Id, ADR(StackArray), TotalElementsStack, PositionFound);
	IF CheckResult <> 0 THEN
		RemoveItemInStack := CheckResult;
		RETURN;
	END_IF

	//Make space in Stack
	ShiftArrayOffset(ADR(StackArray), SIZEOF(StackArray), SIZEOF(StackArray[0]), PositionFound+1, PositionFound, TotalElementsStack - PositionFound -1);

	// Manage Stack index
	TotalElementsStack := TotalElementsStack - 1;

	// Clean values from end
	RemoveItemInStack := CleanEndArray(ADR(StackArray), SIZEOF(StackArray), SIZEOF(StackArray[0]), TotalElementsStack);
	IF RemoveItemInStack <> 0 THEN
		RETURN;
	END_IF

	RemoveItemInStack := 0;

END_FUNCTION
```

#### CheckMedia.st
```iecst
(* Review if the values in a trackignArray is consistent. Using USINT array to load differente lines *)
FUNCTION CheckFilteredMediaLine

	xFilteredData := TRUE;
	//Creating mask with bit active in the right position and invert
	bitLine:=1;
	bitLine := SHL(bitLine,indexLine);
	FOR iIndexArray := sensorPosition TO sensorPosition + mediaFilter DO
		// If the corresponding bit is false, the filter is not matched
		IF (valuesTracking[iIndexArray] AND bitLine) = 0 THEN
			xFilteredData := FALSE;
			EXIT;
		END_IF
	END_FOR
	CheckFilteredMediaLine := xFilteredData;

END_FUNCTION

(* Review if the values in a trackignArray is consistent. Using BOOL array to load individual data *)
FUNCTION CheckFilteredMediaBool

	xFilteredData := TRUE;
	FOR iIndexArray := sensorPosition TO sensorPosition + mediaFilter DO
		// If the corresponding bit is false, the filter is not matched
		IF NOT valuesTracking[iIndexArray] THEN
			xFilteredData := FALSE;
			EXIT;
		END_IF
	END_FOR
	CheckFilteredMediaBool := xFilteredData;

END_FUNCTION
```

#### TrackingEvents.st
```iecst
FUNCTION AddMediaTrackingEvents

	// Moving the array to the right
	ShiftArrayForward(pEventsTrackingArray, SIZEOF(fakeElement) * THICK_MAX_TRACKING_EVENTS, SIZEOF(fakeElement), 1, THICK_MAX_TRACKING_EVENTS-1);

	EventsArray ACCESS(pEventsTrackingArray);
	EventsArray[0].diBeltPosition := diBeltPosition;
	EventsArray[0].diDistanceToPrevious := diBeltPosition - EventsArray[1].diBeltPosition;
	EventsArray[0].Event := EventType;

	AddMediaTrackingEvents := TRUE;

END_FUNCTION
```

### Program Logical/ExtPack/_Media/ThicknessCtrl/ThicknessCtrl_v2/ThicknessCtrl (IEC) - Thickness array analog sensor

#### Alarms.st
```iecst
ACTION Alarms:

	dataHeigh.Alarms.xNoThicknessInstalled 	:= NOT (gDing.State.xDingInstalled OR gPhotoCells.status.xInstalled);

END_ACTION
```

#### AlarmSounds.st
```iecst
ACTION AlarmSounds:

	FOR iIndexCheck:=1 TO MAX_LAST_CHECKMEDIA DO
		ars_CheckMedia[iIndexCheck].xAlarm:= dataHeigh.Alarms.CheckMedia[iIndexCheck];
		ars_CheckMedia[iIndexCheck].xSilence:= dataHeigh.Commands.xMute;
		ars_CheckMedia[iIndexCheck]();
	END_FOR

	ars_NoThicknessSystemInstalled.xAlarm:= dataHeigh.Alarms.xNoThicknessInstalled;
	ars_NoThicknessSystemInstalled.xSilence:= dataHeigh.Commands.xMute;
	ars_NoThicknessSystemInstalled();

	iReasonSound.0 := ars_CheckMedia[1].xAlarmSound;
	iReasonSound.1 := ars_CheckMedia[2].xAlarmSound;
	iReasonSound.2 := ars_NoThicknessSystemInstalled.xAlarmSound;
	dataHeigh.AlSummary.xAlarmSound := iReasonSound > 0;

END_ACTION
```

#### CureTracking.st
```iecst
ACTION RunCureArray:

	//Need to run the matrix through iLastPosition, the max position of the LED
	ShiftArrayForward(ADR(xCuringTracking), SIZEOF(xCuringTracking), SIZEOF(xCuringTracking[0]), iPositionsToRunArray, iLastPosition);

	//Load data depending on the source of the media
	LoadCureMediaFromTrackingMedia;

END_ACTION

ACTION LoadCureMediaFromTrackingMedia:

	IF dataHeigh.status.xNewMediaStackEnabled THEN
		LoadCureMediaFromTrackingMediaStack;
	ELSE
		LoadCureMediaFromTrackingMediaContinuous;
	END_IF

END_ACTION

ACTION LoadCureMediaFromTrackingMediaContinuous:

	// Fill-in moved spaces with data from TrackingMedia.
	// The clean area of Tracking media filtered starts in iSensorPosition + iMediaFilter  + iPositionsToRunArray
	//to be sure that the Tracking media has been cleaned after a end of board slower than the filter
	iProdDetectFilterStartIndex := iProductDetectSensorPosition + dataHeigh.parameters.Detection.ProductDetect.iMediaFilter + iPositionsToRunArray;
	FOR iIndexArray := iProdDetectFilterStartIndex TO iProdDetectFilterStartIndex + iPositionsToRunArray DO //Adding extra values to check
		// Line L1
		xCuringTracking[iIndexArray].INDEXCURING_L1_COLOR := xMediaTracking[iIndexArray].INDEXTRACKING_L1;
		xCuringTracking[iIndexArray].INDEXCURING_L1_WHITE := xMediaTracking[iIndexArray].INDEXTRACKING_L1 AND EnteringMediaContinuous.Media.xHasWhite;
		xCuringTracking[iIndexArray].INDEXCURING_L1_PRIMER := xMediaTracking[iIndexArray].INDEXTRACKING_L1 AND EnteringMediaContinuous.Media.xHasClear;
	END_FOR

	IF NOT dataHeigh.parameters.xDoubleLine THEN
		RETURN;
	END_IF
	FOR iIndexArray := iProdDetectFilterStartIndex TO iProdDetectFilterStartIndex + iPositionsToRunArray DO //Adding extra values to check
		// Line L2
		xCuringTracking[iIndexArray].INDEXCURING_L2_COLOR := xMediaTracking[iIndexArray].INDEXTRACKING_L2;
		xCuringTracking[iIndexArray].INDEXCURING_L2_WHITE := xMediaTracking[iIndexArray].INDEXTRACKING_L2 AND EnteringMediaContinuous.Media.xHasWhite;
		xCuringTracking[iIndexArray].INDEXCURING_L2_PRIMER := xMediaTracking[iIndexArray].INDEXTRACKING_L2 AND EnteringMediaContinuous.Media.xHasClear;
	END_FOR

END_ACTION

ACTION LoadCureMediaFromTrackingMediaStack:

	LoadCureMediaFromTrackingMediaL1;
	IF dataHeigh.parameters.xDoubleLine THEN
		LoadCureMediaFromTrackingMediaL2;
	END_IF

END_ACTION

ACTION LoadCureMediaFromTrackingMediaL1:

	IF MediaTracking_iTotalInsideL1 = 0 THEN
		RETURN;
	END_IF

	// Fill-in moved spaces with data from TrackingMedia.
	// The clean area of Tracking media filtered starts in iSensorPosition + iMediaFilter  + iPositionsToRunArray
	//to be sure that the Tracking media has been cleaned after a end of board slower than the filter
	iProdDetectFilterStartIndex := iProductDetectSensorPosition + dataHeigh.parameters.Detection.ProductDetect.iMediaFilter  + THICK_MAX_UPDATE_VALUES + iPositionsToRunArray;
	xDetectedGap_L1 := FALSE;
	FOR iIndexArray := iProdDetectFilterStartIndex TO iProdDetectFilterStartIndex + iPositionsToRunArray DO //Adding extra values to check

		// Line L1
		IF NOT xDetectedGap_L1 THEN
			xCuringTracking[iIndexArray].INDEXCURING_L1_COLOR := xMediaTracking[iIndexArray].INDEXTRACKING_L1;
			xCuringTracking[iIndexArray].INDEXCURING_L1_WHITE := xMediaTracking[iIndexArray].INDEXTRACKING_L1 AND EnteringMediaL1.Media.xHasWhite;
			xCuringTracking[iIndexArray].INDEXCURING_L1_PRIMER := xMediaTracking[iIndexArray].INDEXTRACKING_L1 AND EnteringMediaContinuous.Media.xHasClear;
		ELSE
			IF MediaTracking_iTotalInsideL1 >= 2 THEN
				xCuringTracking[iIndexArray].INDEXCURING_L1_COLOR := xMediaTracking[iIndexArray].INDEXTRACKING_L1;
				xCuringTracking[iIndexArray].INDEXCURING_L1_WHITE := xMediaTracking[iIndexArray].INDEXTRACKING_L1 AND MediaTrackingInsideL1[MediaTracking_iTotalInsideL1-2].Media.xHasWhite;
				xCuringTracking[iIndexArray].INDEXCURING_L1_PRIMER := xMediaTracking[iIndexArray].INDEXTRACKING_L1 AND MediaTrackingInsideL1[MediaTracking_iTotalInsideL1-2].Media.xHasClear;
			END_IF
		END_IF

		//Detecting the gap inside the positions to tun
		IF xMediaTracking[iIndexArray].INDEXTRACKING_L1 AND NOT xMediaTracking[iIndexArray+1].INDEXTRACKING_L1 THEN xDetectedGap_L1 := TRUE; END_IF

	END_FOR

END_ACTION

ACTION LoadCureMediaFromTrackingMediaL2:

	IF MediaTracking_iTotalInsideL2 = 0 THEN
		RETURN;
	END_IF

	// Fill-in moved spaces with data from TrackingMedia.
	// The clean area of Tracking media filtered starts in iSensorPosition + iMediaFilter  + iPositionsToRunArray
	//to be sure that the Tracking media has been cleaned after a end of board slower than the filter
	iProdDetectFilterStartIndex := iProductDetectSensorPosition + dataHeigh.parameters.Detection.ProductDetect.iMediaFilter + iPositionsToRunArray;
	xDetectedGap_L2 := FALSE;
	FOR iIndexArray := iProdDetectFilterStartIndex TO iProdDetectFilterStartIndex + iPositionsToRunArray DO //Adding extra values to check

		// Line L2
		IF NOT xDetectedGap_L2 THEN
			xCuringTracking[iIndexArray].INDEXCURING_L2_COLOR := xMediaTracking[iIndexArray].INDEXTRACKING_L2;
			xCuringTracking[iIndexArray].INDEXCURING_L2_WHITE := xMediaTracking[iIndexArray].INDEXTRACKING_L2 AND EnteringMediaL2.Media.xHasWhite;
			xCuringTracking[iIndexArray].INDEXCURING_L2_PRIMER := xMediaTracking[iIndexArray].INDEXTRACKING_L2 AND EnteringMediaL2.Media.xHasClear;
		ELSE
			IF MediaTracking_iTotalInsideL2 >= 2 THEN
				xCuringTracking[iIndexArray].INDEXCURING_L2_COLOR := xMediaTracking[iIndexArray].INDEXTRACKING_L2;
				xCuringTracking[iIndexArray].INDEXCURING_L2_WHITE := xMediaTracking[iIndexArray].INDEXTRACKING_L2 AND MediaTrackingInsideL2[MediaTracking_iTotalInsideL2-2].Media.xHasWhite;
				xCuringTracking[iIndexArray].INDEXCURING_L2_PRIMER := xMediaTracking[iIndexArray].INDEXTRACKING_L2 AND MediaTrackingInsideL2[MediaTracking_iTotalInsideL2-2].Media.xHasClear;
			END_IF
		END_IF

		//Detecting the gap inside the positions to tun
		IF xMediaTracking[iIndexArray].INDEXTRACKING_L2 AND NOT xMediaTracking[iIndexArray+1].INDEXTRACKING_L2 THEN xDetectedGap_L2 := TRUE; END_IF

	END_FOR

END_ACTION

ACTION ReviewCuringActivation:

	//White
	CureLampParams ACCESS ADR(dataHeigh.parameters.Cure.White);
	IF CureLampParams.xEnabled THEN
		iStartCuringWindow := LIMIT(1, CureLampParams.iStartWindow, iMAXTRACKINGARRAY);
		iEndCuringWindow := LIMIT(1, CureLampParams.iEndWindow, iMAXTRACKINGARRAY);
		IF NOT dataHeigh.parameters.Cure.xEnableMediaTracking THEN
			ReviewCuringActivationWhite;
		ELSE
			dataHeigh.status.MediaPosition.L1.White.xMediaInLedPosition := ReviewMediaTrackingInPosition(ADR(MediaTrackingInsideL1), MediaTracking_iTotalInsideL1, iStartCuringWindow, iEndCuringWindow, TRUE);
			IF dataHeigh.parameters.xDoubleLine THEN
				dataHeigh.status.MediaPosition.L2.White.xMediaInLedPosition := ReviewMediaTrackingInPosition(ADR(MediaTrackingInsideL2), MediaTracking_iTotalInsideL2, iStartCuringWindow, iEndCuringWindow, TRUE);
			END_IF

		END_IF
	END_IF

	//Color
	CureLampParams ACCESS ADR(dataHeigh.parameters.Cure.Color);
	IF CureLampParams.xEnabled THEN
		iStartCuringWindow := LIMIT(1, CureLampParams.iStartWindow, iMAXTRACKINGARRAY);
		iEndCuringWindow := LIMIT(1, CureLampParams.iEndWindow, iMAXTRACKINGARRAY);
		IF NOT dataHeigh.parameters.Cure.xEnableMediaTracking THEN
			ReviewCuringActivationColor;
		ELSE
			dataHeigh.status.MediaPosition.L1.Color.xMediaInLedPosition := ReviewMediaTrackingInPosition(ADR(MediaTrackingInsideL1), MediaTracking_iTotalInsideL1, iStartCuringWindow, iEndCuringWindow, FALSE);
			IF dataHeigh.parameters.xDoubleLine THEN
				dataHeigh.status.MediaPosition.L2.Color.xMediaInLedPosition := ReviewMediaTrackingInPosition(ADR(MediaTrackingInsideL2), MediaTracking_iTotalInsideL2, iStartCuringWindow, iEndCuringWindow, FALSE);
			END_IF
		END_IF
	END_IF

	//Primer
	CureLampParams ACCESS ADR(dataHeigh.parameters.Cure.Primer);
	IF CureLampParams.xEnabled THEN
		iStartCuringWindow := LIMIT(1, CureLampParams.iStartWindow, iMAXTRACKINGARRAY);
		iEndCuringWindow := LIMIT(1, CureLampParams.iEndWindow, iMAXTRACKINGARRAY);
		IF NOT dataHeigh.parameters.Cure.xEnableMediaTracking THEN
			ReviewCuringActivationPrimer;
		ELSE
			dataHeigh.status.MediaPosition.L1.Primer.xMediaInLedPosition := ReviewMediaTrackingInPosition(ADR(MediaTrackingInsideL1), MediaTracking_iTotalInsideL1, iStartCuringWindow, iEndCuringWindow, FALSE);
			IF dataHeigh.parameters.xDoubleLine THEN
				dataHeigh.status.MediaPosition.L2.Primer.xMediaInLedPosition := ReviewMediaTrackingInPosition(ADR(MediaTrackingInsideL2), MediaTracking_iTotalInsideL2, iStartCuringWindow, iEndCuringWindow, FALSE);
			END_IF
		END_IF
	END_IF
END_ACTION

ACTION ReviewCuringActivationWhite:

	ReviewCuringActivationWhiteL1;
	IF dataHeigh.parameters.xDoubleLine THEN
		ReviewCuringActivationWhiteL2;
	END_IF

END_ACTION

ACTION ReviewCuringActivationWhiteL1:

	xMediaInLedPositionWhiteL1 := FALSE;
	FOR iIndexWindow := iStartCuringWindow TO iEndCuringWindow DO
		IF xCuringTracking[iIndexWindow].INDEXCURING_L1_WHITE THEN
			xMediaInLedPositionWhiteL1 := TRUE;
			EXIT;
		END_IF
	END_FOR
	dataHeigh.status.MediaPosition.L1.White.xMediaInLedPosition := xMediaInLedPositionWhiteL1;

END_ACTION

ACTION ReviewCuringActivationWhiteL2:

	xMediaInLedPositionWhiteL2 := FALSE;
	FOR iIndexWindow := iStartCuringWindow TO iEndCuringWindow DO
		IF xCuringTracking[iIndexWindow].INDEXCURING_L2_WHITE THEN
			xMediaInLedPositionWhiteL2 := TRUE;
			EXIT;
		END_IF
	END_FOR
	dataHeigh.status.MediaPosition.L2.White.xMediaInLedPosition := xMediaInLedPositionWhiteL2;

END_ACTION

ACTION ReviewCuringActivationColor:

	ReviewCuringActivationColorL1;
	IF dataHeigh.parameters.xDoubleLine THEN
		ReviewCuringActivationColorL2;
	END_IF

END_ACTION

ACTION ReviewCuringActivationColorL1:

	xMediaInLedPositionColorL1 := FALSE;
	FOR iIndexWindow := iStartCuringWindow TO iEndCuringWindow DO
		IF xCuringTracking[iIndexWindow].INDEXCURING_L1_COLOR THEN
			xMediaInLedPositionColorL1 := TRUE;
			EXIT;
		END_IF
	END_FOR
	dataHeigh.status.MediaPosition.L1.Color.xMediaInLedPosition := xMediaInLedPositionColorL1;

END_ACTION

ACTION ReviewCuringActivationColorL2:

	xMediaInLedPositionColorL2 := FALSE;
	FOR iIndexWindow := iStartCuringWindow TO iEndCuringWindow DO
		IF xCuringTracking[iIndexWindow].INDEXCURING_L2_COLOR THEN
			xMediaInLedPositionColorL2 := TRUE;
			EXIT;
		END_IF
	END_FOR
	dataHeigh.status.MediaPosition.L2.Color.xMediaInLedPosition := xMediaInLedPositionColorL2;

END_ACTION

ACTION ReviewCuringActivationPrimer:

	ReviewCuringActivationPrimerL1;
	IF dataHeigh.parameters.xDoubleLine THEN
		ReviewCuringActivationPrimerL2;
	END_IF

END_ACTION

ACTION ReviewCuringActivationPrimerL1:

	xMediaInLedPositionPrimerL1 := FALSE;
	FOR iIndexWindow := iStartCuringWindow TO iEndCuringWindow DO
		IF xCuringTracking[iIndexWindow].INDEXCURING_L1_PRIMER THEN
			xMediaInLedPositionPrimerL1 := TRUE;
			EXIT;
		END_IF
	END_FOR
	dataHeigh.status.MediaPosition.L1.Primer.xMediaInLedPosition := xMediaInLedPositionPrimerL1;

END_ACTION

ACTION ReviewCuringActivationPrimerL2:

	xMediaInLedPositionPrimerL2 := FALSE;
	FOR iIndexWindow := iStartCuringWindow TO iEndCuringWindow DO
		IF xCuringTracking[iIndexWindow].INDEXCURING_L2_PRIMER THEN
			xMediaInLedPositionPrimerL2 := TRUE;
			EXIT;
		END_IF
	END_FOR
	dataHeigh.status.MediaPosition.L2.Primer.xMediaInLedPosition := xMediaInLedPositionPrimerL2;

END_ACTION
```

#### DryTracking.st
```iecst
ACTION ReviewDryActivation:

	// Limit the value configured relative to power reductions
	rSubstratePowerReduction := LIMIT(0.3 , dataHeigh.parameters.Dry.rSubstratePowerReduction, 1);
	rThermalInerciaReduction := LIMIT(0.6 , dataHeigh.parameters.Dry.rThermalInerciaReduction, 1);
	rPowerReduction := rSubstratePowerReduction * rThermalInerciaReduction;

	iDistanceDelay := REAL_TO_UINT(dataHeigh.parameters.Dry.rCommsDelay * dataHeigh.parameters.Belt.rBeltSpeed / 600.0);
	iDistanceWindow := REAL_TO_UINT((dataHeigh.parameters.Dry.rThermalDelay + dataHeigh.parameters.Dry.rCommsDelay) * dataHeigh.parameters.Belt.rBeltSpeed / 600.0);

	// IntensityPower for Lamps in L1
	FOR iIndexDryer := 1 TO MAX_LAST_NIR_MODULES DO

		DryerInfo ACCESS ADR(dataHeigh.parameters.Dry.Dryers[iIndexDryer]);

		iEndCuringWindow := LIMIT(1, DryerInfo.iPosition - iDistanceDelay, iMAXTRACKINGARRAY);
		// Assure the start window remains in positive values
		iStartCuringWindow := UINT_TO_INT(iEndCuringWindow) - UINT_TO_INT(iDistanceWindow);

		RevMediaTrackingEnergyInPos(ADR(MediaTrackingInsideL1),
										MediaTracking_iTotalInsideL1,
										iStartCuringWindow,
										iEndCuringWindow,
										dataHeigh.parameters.Dry.iLamps,
										dataHeigh.parameters.Dry.rLampWidth,
										dataHeigh.parameters.Dry.rLampOffset,
										dataHeigh.parameters.Dry.rDryExtend,
										dataHeigh.parameters.Dry.iMinDryValue,
										dataHeigh.status.MediaPosition.L1.NirDryer[iIndexDryer].Intensity);
	END_FOR

	// If simple line, assign L1 to total and return
	IF NOT dataHeigh.parameters.xDoubleLine THEN
		dataHeigh.status.Dry[1].Intensity := dataHeigh.status.MediaPosition.L1.NirDryer[1].Intensity;
		dataHeigh.status.Dry[2].Intensity := dataHeigh.status.MediaPosition.L1.NirDryer[2].Intensity;
		RETURN;
	END_IF

	// IntensityPower for Lamps in L2
	FOR iIndexDryer := 1 TO MAX_LAST_NIR_MODULES DO

		DryerInfo ACCESS ADR(dataHeigh.parameters.Dry.Dryers[iIndexDryer]);

		iEndCuringWindow := LIMIT(1, DryerInfo.iPosition - iDistanceDelay, iMAXTRACKINGARRAY);
		iStartCuringWindow := LIMIT(1, iEndCuringWindow - iDistanceDelay, iMAXTRACKINGARRAY);

		RevMediaTrackingEnergyInPos(ADR(MediaTrackingInsideL2),
										MediaTracking_iTotalInsideL2,
										iStartCuringWindow,
										iEndCuringWindow,
										dataHeigh.parameters.Dry.iLamps,
										dataHeigh.parameters.Dry.rLampWidth,
										dataHeigh.parameters.Dry.rLampOffset,
										dataHeigh.parameters.Dry.rDryExtend,
										dataHeigh.parameters.Dry.iMinDryValue,
										dataHeigh.status.MediaPosition.L2.NirDryer[iIndexDryer].Intensity);
	END_FOR

	// Assigning data from each line to the Intensity status of each dryer
	FOR iIndexArray := 1 TO THICKENERGY_MAX_LAMPS DO
		dataHeigh.status.Dry[1].Intensity[iIndexArray] := REAL_TO_INT( rPowerReduction * MAX(dataHeigh.status.MediaPosition.L1.NirDryer[1].Intensity[iIndexArray], dataHeigh.status.MediaPosition.L2.NirDryer[1].Intensity[iIndexArray]) );
		dataHeigh.status.Dry[2].Intensity[iIndexArray] := REAL_TO_INT( rPowerReduction * MAX(dataHeigh.status.MediaPosition.L1.NirDryer[2].Intensity[iIndexArray], dataHeigh.status.MediaPosition.L2.NirDryer[2].Intensity[iIndexArray]) );
	END_FOR

END_ACTION

// Calling outside the running belt code
ACTION ReviewDryManual:

	// Temporaty while DDC dynamic is not active
	IF EDGEPOS(dataHeigh.parameters.AutoMode.xProduction) THEN
		dataHeigh.parSw.Dry.xGetMaxFromFileInfo := TRUE;
	END_IF

	IF EDGEPOS(dataHeigh.parSw.Dry.xGetMaxFromFileInfo) THEN
		FOR iIndexArray := 1 TO THICKENERGY_MAX_LAMPS DO
			MaxLampIntensityL1[iIndexArray] := 0;
			MaxLampIntensityL2[iIndexArray] := 0;
		END_FOR
	END_IF
	// Calculating the max of the file information
	IF dataHeigh.parSw.Dry.xGetMaxFromFileInfo THEN
		FOR iIndexArray := 1 TO THICKENERGY_MAX_LAMPS DO
			MaxLampIntensityL1[iIndexArray] := MAX(MaxLampIntensityL1[iIndexArray] , dataHeigh.status.MediaPosition.L1.NirDryer[1].Intensity[iIndexArray], dataHeigh.parameters.Dry.iMinDryValue);
			MaxLampIntensityL2[iIndexArray] := MAX(MaxLampIntensityL2[iIndexArray] , dataHeigh.status.MediaPosition.L1.NirDryer[2].Intensity[iIndexArray], dataHeigh.parameters.Dry.iMinDryValue);
		END_FOR
	END_IF

	IF dataHeigh.parSw.Dry.xGetMaxFromFileInfo AND (xExitingMediaL1 OR EDGEPOS(dataHeigh.status.Belt.xBeltEmpty)) THEN
		dataHeigh.parSw.Dry.ManIntensity[1].Intensity := MaxLampIntensityL1;
		dataHeigh.parSw.Dry.ManIntensity[2].Intensity := MaxLampIntensityL2;
		dataHeigh.parSw.Dry.xGetMaxFromFileInfo := FALSE;
	END_IF

	IF dataHeigh.parSw.Dry.xForceManIntensity THEN
		dataHeigh.status.Dry := dataHeigh.parSw.Dry.ManIntensity;
	END_IF

END_ACTION
```

#### MediaTracking.st
```iecst
ACTION RunMediaArray:

	//Need to run the matrix through all belts
	ShiftArrayForward(ADR(xMediaTracking), SIZEOF(xMediaTracking), SIZEOF(xMediaTracking[0]), iPositionsToRunArray, iMaxTrackingPosition + THICK_MAX_UPDATE_VALUES); //Ading extra values to allow view the edges for exiting

	//Load data depending on the source of the media
	IF dataHeigh.parameters.Detection.ProductDetect.xLoadMedia THEN
		LoadAndCheckMediaFromProductDetectL1;
		IF dataHeigh.parameters.xDoubleLine THEN
			LoadAndCheckMediaFromProductDetectL2;
		END_IF
		// Using the Inside arrays just if Curing or Drying is enabled in tracking
		IF dataHeigh.status.xMediaTrackingEnabled THEN
			iSensorFilterStartIndex := iProductDetectSensorPosition + dataHeigh.parameters.Detection.ProductDetect.iMediaFilter;
			CheckFinishEnteringMedia;
			iSensorFilterStartIndex := iProductDetectSensorPosition + dataHeigh.parameters.Detection.ProductDetect.iMediaFilter;
			CheckEnteringMedia;
		END_IF
	END_IF

	// Allow the detection from the arraySensors independent of if it is used to load main data
	IF gPhotoCells.status.xInstalled THEN
		//Calculating number of positions to be updated
		iNumberOfPositionsToBeUpdated := dataHeigh.parameters.Detection.Array.iMediaFilter + THICK_MAX_UPDATE_VALUES;
		IF dataHeigh.Commands.xReviewIncoherenceArrayAndPd THEN
			iNumberOfPositionsToBeUpdated := iNumberOfPositionsToBeUpdated + dataHeigh.parameters.iDistanceFromArrayToPd;
		END_IF
		ShiftArrayForward(ADR(xMediaPresentArray), SIZEOF(xMediaPresentArray), SIZEOF(xMediaPresentArray[0]), iPositionsToRunArray, iNumberOfPositionsToBeUpdated);

		LoadMediaFromArraySensor;

		IF dataHeigh.parameters.Detection.Array.xLoadMedia THEN
			CheckFilteredArraySensorMedia;
		END_IF

		IF dataHeigh.parameters.Detection.Array.xEnableSensorIncoherAlarm THEN
			SensorsArrayAndProductDetectIncoherence;
		END_IF
	END_IF

	IF dataHeigh.parameters.Detection.Analog.xLoadMedia AND gDing.State.xDingInstalled THEN
		//Calculating number of positions to be updated
		iNumberOfPositionsToBeUpdated := dataHeigh.parameters.Detection.Analog.iMediaFilter + THICK_MAX_UPDATE_VALUES;

		ShiftArrayForward(ADR(xMediaPresentAnalog), SIZEOF(xMediaPresentAnalog), SIZEOF(xMediaPresentAnalog[0]), iPositionsToRunArray, iNumberOfPositionsToBeUpdated);
		LoadMediaFromAnalogSensor;
		CheckFilteredAnalogSensorMedia;
	END_IF

	IF dataHeigh.parameters.Detection.Basic.xLoadMedia AND gBasicDetectMedia.Status.xInstalled THEN
		//Calculating number of positions to be updated
		iNumberOfPositionsToBeUpdated := dataHeigh.parameters.Detection.Basic.iMediaFilter + THICK_MAX_UPDATE_VALUES;

		ShiftArrayForward(ADR(xMediaPresentBasic), SIZEOF(xMediaPresentBasic), SIZEOF(xMediaPresentBasic[0]), iPositionsToRunArray, iNumberOfPositionsToBeUpdated);
		LoadMediaFromBasicDetectMedia;

		// MediaTracking can just be loaded from one source data
		IF dataHeigh.parameters.Detection.Basic.xEnableMediaTracking AND NOT dataHeigh.parameters.Detection.ProductDetect.xLoadMedia THEN
			// Load the data from Basic into MediaTracking to allow working with internal arrays of media inside the machine
			LoadMediaFromFastDataLine(ADR(dataHeigh.Internal.MediaDetectionValuesL1), dataHeigh.Internal.rFastValues, INDEXTRACKING_L1, iPositionsToRunArray, dataHeigh.parameters.Detection.Basic.iSensorPosition, ADR(xMediaTracking));
			IF dataHeigh.parameters.xDoubleLine THEN
				LoadMediaFromFastDataLine(ADR(dataHeigh.Internal.MediaDetectionValuesL2), dataHeigh.Internal.rFastValues, INDEXTRACKING_L2, iPositionsToRunArray, dataHeigh.parameters.Detection.Basic.iSensorPosition, ADR(xMediaTracking));
			END_IF
			// Loading media with Basic just if there is no ProductDetec (mainly in Dryer)
			IF dataHeigh.status.xMediaTrackingEnabled THEN
				iSensorFilterStartIndex := dataHeigh.parameters.Detection.Basic.iSensorPosition + dataHeigh.parameters.Detection.Basic.iMediaFilter;
				CheckFinishEnteringMedia;
				iSensorFilterStartIndex := dataHeigh.parameters.Detection.Basic.iSensorPosition + dataHeigh.parameters.Detection.Basic.iMediaFilter;
				CheckEnteringMedia;
			END_IF
		END_IF
		CheckFilteredBasicDetectionMedia;
	END_IF

	dataHeigh.Outputs.xMediaFiltered := xFilteredProductDetectMediaL1 OR xFilteredProductDetectMediaL2 OR xFilteredArraySensorMedia OR xFilteredAnalogSensorMedia OR xFilteredBasicDetectionMedia;

	// In case any tracking active, RUN and check exiting
	IF dataHeigh.status.xMediaTrackingEnabled THEN
		RunMediaInsidePositions;
		CheckExitingMedia;
	END_IF

	MediaTracking_xEnteringMachineL1 := MediaTracking_iTotalInsideL1>MediaTracking_iTotalInsideL1_cp;
	MediaTracking_xEnteringMachineL2 := MediaTracking_iTotalInsideL2>MediaTracking_iTotalInsideL2_cp;
	MediaTracking_iTotalInsideL1_cp := MediaTracking_iTotalInsideL1;
	MediaTracking_iTotalInsideL2_cp := MediaTracking_iTotalInsideL2;

END_ACTION

ACTION LoadAndCheckMediaFromProductDetectL1:
	LoadMediaFromProductDetectL1;
	CheckAndCleanProductDetectMediaFilterL1;
	CheckFilteredProductDetectMediaL1;
END_ACTION

ACTION LoadAndCheckMediaFromProductDetectL2:
	LoadMediaFromProductDetectL2;
	CheckAndCleanProductDetectMediaFilterL2;
	CheckFilteredProductDetectMediaL2;
END_ACTION

ACTION LoadMediaFromProductDetectL1:

	LoadMediaFromFastDataLine(ADR(dataHeigh.Internal.ProductDetectValuesL1), dataHeigh.Internal.rFastValues, INDEXTRACKING_L1, iPositionsToRunArray, iProductDetectSensorPosition, ADR(xMediaTracking));

END_ACTION

ACTION LoadMediaFromProductDetectL2:

	LoadMediaFromFastDataLine(ADR(dataHeigh.Internal.ProductDetectValuesL2), dataHeigh.Internal.rFastValues, INDEXTRACKING_L2, iPositionsToRunArray, iProductDetectSensorPosition, ADR(xMediaTracking));

END_ACTION

ACTION LoadMediaFromAnalogSensor:

	LoadMediaFromFastDataBool(ADR(dataHeigh.Internal.MediaAnalogValues), dataHeigh.Internal.rFastValues, iPositionsToRunArray, 0, ADR(xMediaPresentAnalog));

END_ACTION

ACTION LoadMediaFromArraySensor:

	LoadMediaFromFastDataBool(ADR(dataHeigh.Internal.MediaArraySensorValues), dataHeigh.Internal.rFastValues, iPositionsToRunArray, 0, ADR(xMediaPresentArray));

END_ACTION

ACTION LoadMediaFromBasicDetectMedia:

	LoadMediaFromFastDataBool(ADR(dataHeigh.Internal.MediaDetectionValues), dataHeigh.Internal.rFastValues, iPositionsToRunArray, 0, ADR(xMediaPresentBasic));

END_ACTION

ACTION CheckFilteredProductDetectMediaL1:

	xFilteredProductDetectMediaL1 := CheckFilteredMediaLine(ADR(xMediaTracking), INDEXTRACKING_L1, iProductDetectSensorPosition, dataHeigh.parameters.Detection.ProductDetect.iMediaFilter);
	dataHeigh.status.Detection.xFilteredProductDetectMediaL1 := xFilteredProductDetectMediaL1;

END_ACTION

ACTION CheckFilteredProductDetectMediaL2:

	xFilteredProductDetectMediaL2 := CheckFilteredMediaLine(ADR(xMediaTracking), INDEXTRACKING_L2, iProductDetectSensorPosition, dataHeigh.parameters.Detection.ProductDetect.iMediaFilter);
	dataHeigh.status.Detection.xFilteredProductDetectMediaL2 := xFilteredProductDetectMediaL2;

END_ACTION

ACTION CheckFilteredAnalogSensorMedia:

	xFilteredAnalogSensorMedia := CheckFilteredMediaBool(ADR(xMediaPresentAnalog), 0, dataHeigh.parameters.Detection.Analog.iMediaFilter);
	dataHeigh.status.Detection.xFilteredAnalogSensorMedia := xFilteredAnalogSensorMedia;

END_ACTION

ACTION CheckFilteredArraySensorMedia:

	xFilteredArraySensorMedia := CheckFilteredMediaBool(ADR(xMediaPresentArray), 0, dataHeigh.parameters.Detection.Array.iMediaFilter);
	dataHeigh.status.Detection.xFilteredArraySensorMedia := xFilteredArraySensorMedia;

END_ACTION

ACTION CheckFilteredBasicDetectionMedia:

	xFilteredBasicDetectionMedia := CheckFilteredMediaBool(ADR(xMediaPresentBasic), 0, dataHeigh.parameters.Detection.Basic.iMediaFilter);
	dataHeigh.status.Detection.xFilteredBasicDetectionMedia := xFilteredBasicDetectionMedia;

END_ACTION

ACTION CheckAndCleanProductDetectMediaFilterL1:

	// With a 0, filter is disabled
	IF dataHeigh.parameters.Detection.ProductDetect.iMediaFilter = 0 THEN
		RETURN;
	END_IF

	//Starting from the sensor position and reviewing for each end of board if the new board in consistent enough
	iProdDetectFilterStartIndex := iProductDetectSensorPosition;

	FOR iIndexArray := iProdDetectFilterStartIndex TO iProdDetectFilterStartIndex + iPositionsToRunArray + 1 DO

		// Detecting the end of a board.
		// If using the Filter while detecting the start of a board, the end of previous board with small gap can be "cleaned" and would be an error
		IF NOT xMediaTracking[iIndexArray].INDEXTRACKING_L1 AND xMediaTracking[iIndexArray + 1].INDEXTRACKING_L1 THEN
			// Going for the end of the filter. All data has to be true
			// Starting in (iIndexArray + 1) to start checking in TRUE values
			FOR iIndexNewMediaArray := iIndexArray + 1 TO iIndexArray + dataHeigh.parameters.Detection.ProductDetect.iMediaFilter + 1 DO
				//If reading a 0 is because signal is not robust
				IF NOT xMediaTracking[iIndexNewMediaArray].INDEXTRACKING_L1 THEN
					//Clean al data for the false pulse
					FOR iIndexCleanMediaArray := iIndexNewMediaArray TO iIndexArray BY -1 DO
						xMediaTracking[iIndexCleanMediaArray].INDEXTRACKING_L1 := FALSE;
					END_FOR
					EXIT; //The filter has not been validated, so not keep on searching for FALSEs
				END_IF
			END_FOR
		END_IF
	END_FOR

END_ACTION

ACTION CheckAndCleanProductDetectMediaFilterL2:

	// With a 0, filter is disabled
	IF dataHeigh.parameters.Detection.ProductDetect.iMediaFilter = 0 THEN
		RETURN;
	END_IF

	//Starting from the sensor position and reviewing for each end of board if the new board in consistent enough
	iProdDetectFilterStartIndex := iProductDetectSensorPosition;

	FOR iIndexArray := iProdDetectFilterStartIndex TO iProdDetectFilterStartIndex + iPositionsToRunArray + 1 DO

		// Detecting the end of a board.
		// If using the Filter while detecting the start of a board, the end of previos board with small gap can be "cleaned" and would be an error
		IF NOT xMediaTracking[iIndexArray].INDEXTRACKING_L2 AND xMediaTracking[iIndexArray + 1].INDEXTRACKING_L2 THEN
			// Going for the end of the filter. All data has to be true
			// Starting in (iIndexArray + 1) to start checking in TRUE values
			FOR iIndexNewMediaArray := iIndexArray + 1 TO iIndexArray + dataHeigh.parameters.Detection.ProductDetect.iMediaFilter + 1 DO
				//If reading a 0 is because signal is not robust
				IF NOT xMediaTracking[iIndexNewMediaArray].INDEXTRACKING_L2 THEN
					//Clean al data for the false pulse
					FOR iIndexCleanMediaArray := iIndexNewMediaArray TO iIndexArray BY -1 DO
						xMediaTracking[iIndexCleanMediaArray].INDEXTRACKING_L2 := FALSE;
					END_FOR
					EXIT; //The filter has not been validated, so not keep on searching for FALSEs
				END_IF
			END_FOR
		END_IF
	END_FOR

END_ACTION

(* Needs to be called updating the value of iSensorFilterStartIndex in the form: iSensorFilterStartIndex := iXXXXSensorPosition + dataHeigh.parameters.Detection.XXXXX.iMediaFilter  *)
ACTION CheckEnteringMedia:

	// Old code. This assignation has to be done before calling the ACTION
	//iSensorFilterStartIndex := iProductDetectSensorPosition + dataHeigh.parameters.Detection.ProductDetect.iMediaFilter + THICK_MAX_UPDATE_VALUES;
	// Adding THICK_MAX_UPDATE_VALUES has been removed because it has no sense. Here the index is cm and THICK_MAX_UPDATE_VALUES is data from Fast into Slow

	// Run the exact positions moved to avoid detecting the begining of a board more than once
	FOR iIndexEnteringMedia := iSensorFilterStartIndex TO iSensorFilterStartIndex + iPositionsToRunArray - 1 DO
		// Detecting the start of a board once the filter is full with media
		IF xMediaTracking[iIndexEnteringMedia].INDEXTRACKING_L1 AND NOT xMediaTracking[iIndexEnteringMedia + 1].INDEXTRACKING_L1 THEN
			NewMediaEnteringL1;
			EXIT; //The new board has been detected, so not keep on searching for FALSEs
		END_IF
	END_FOR

	// Run the exact positions moved to avoid detecting the begining of a board more than once
	IF NOT dataHeigh.parameters.xDoubleLine THEN
		RETURN;
	END_IF
	FOR iIndexArray := iSensorFilterStartIndex TO iSensorFilterStartIndex + iPositionsToRunArray -1 DO
		// Detecting the start of a board once the filter is full with media
		IF xMediaTracking[iIndexArray].INDEXTRACKING_L2 AND NOT xMediaTracking[iIndexArray + 1].INDEXTRACKING_L2 THEN
			NewMediaEnteringL2;
			EXIT; //The new board has been detected, so not keep on searching for FALSEs
		END_IF
	END_FOR

END_ACTION

(* Needs to be called updating the value of iSensorFilterStartIndex in the form: iSensorFilterStartIndex := iXXXXSensorPosition + dataHeigh.parameters.Detection.XXXXX.iMediaFilter  *)
ACTION CheckFinishEnteringMedia:

	// Old code. This assignation has to be done before calling the ACTION
	//iSensorFilterStartIndex := iProductDetectSensorPosition + dataHeigh.parameters.Detection.ProductDetect.iMediaFilter + THICK_MAX_UPDATE_VALUES;
	// Adding THICK_MAX_UPDATE_VALUES has been removed because it has no sense. Here the index is cm and THICK_MAX_UPDATE_VALUES is data from Fast into Slow

	// Run the exact positions moved to avoid detecting the begining of a board more than once
	FOR iIndexFinishEnteringMedia := iSensorFilterStartIndex TO iSensorFilterStartIndex + iPositionsToRunArray - 1 DO
		// Detecting the start of a board once the filter is full with media
		IF NOT xMediaTracking[iIndexFinishEnteringMedia].INDEXTRACKING_L1 AND xMediaTracking[iIndexFinishEnteringMedia + 1].INDEXTRACKING_L1 THEN
			FinishEnteringMediaL1;
			EXIT; //The new board has been detected, so not keep on searching for FALSEs
		END_IF
	END_FOR

	// Run the exact positions moved to avoid detecting the begining of a board more than once
	IF NOT dataHeigh.parameters.xDoubleLine THEN
		RETURN;
	END_IF
	FOR iIndexArray := iSensorFilterStartIndex TO iSensorFilterStartIndex + iPositionsToRunArray -1 DO
		// Detecting the start of a board once the filter is full with media
		IF NOT xMediaTracking[iIndexArray].INDEXTRACKING_L2 AND xMediaTracking[iIndexArray + 1].INDEXTRACKING_L2 THEN
			FinishEnteringMediaL2;
			EXIT; //The new board has been detected, so not keep on searching for FALSEs
		END_IF
	END_FOR

END_ACTION

ACTION NewMediaEnteringL1:

	iBoardsBelowBlockL1 := iBoardsBelowBlockL1 + 1;
	dataHeigh.status.Detection.iBoardsFromStartL1 := dataHeigh.status.Detection.iBoardsFromStartL1 + 1;
	dataHeigh.status.Detection.iTotalBoardsL1 := dataHeigh.status.Detection.iTotalBoardsL1 + 1;
	MoveMediaFromNewToInsideL1;
	MediaTracking_iTotalInsideL1; //Just to enable monitor it

END_ACTION

ACTION NewMediaEnteringL2:

	iBoardsBelowBlockL2 := iBoardsBelowBlockL2 + 1;
	dataHeigh.status.Detection.iBoardsFromStartL2 := dataHeigh.status.Detection.iBoardsFromStartL2 + 1;
	dataHeigh.status.Detection.iTotalBoardsL2 := dataHeigh.status.Detection.iTotalBoardsL2 + 1;
	MoveMediaFromNewToInsideL2;
	MediaTracking_iTotalInsideL2; //Just to enable monitor it

END_ACTION

(* Assigning the value of the Tail position of the media   *)
ACTION FinishEnteringMediaL1:

	// Protection if not media inside
	IF MediaTracking_iTotalInsideL1 = 0 THEN
		RETURN;
	END_IF

	IF dataHeigh.parameters.Detection.ProductDetect.xLoadMedia THEN
		MediaTrackingInsideL1[MediaTracking_iTotalInsideL1 - 1].TailPosition := iIndexFinishEnteringMedia;
	ELSIF dataHeigh.parameters.Detection.Basic.xEnableMediaTracking THEN
		MediaTrackingInsideL1[MediaTracking_iTotalInsideL1 - 1].TailPosition := dataHeigh.parameters.Detection.Basic.iSensorPosition + dataHeigh.parameters.Detection.Basic.iMediaFilter;
	END_IF

	AddMediaTrackingEvents(diTotalCmBelt, TAIL_DETECTED, ADR(TrackingEventsArray));

END_ACTION

ACTION FinishEnteringMediaL2:

	// Protection if not media inside
	IF MediaTracking_iTotalInsideL2 = 0 THEN
		RETURN;
	END_IF

	IF dataHeigh.parameters.Detection.ProductDetect.xLoadMedia THEN
		MediaTrackingInsideL1[MediaTracking_iTotalInsideL2 - 1].TailPosition := iProductDetectSensorPosition + dataHeigh.parameters.Detection.ProductDetect.iMediaFilter;
	ELSIF dataHeigh.parameters.Detection.Basic.xEnableMediaTracking THEN
		MediaTrackingInsideL1[MediaTracking_iTotalInsideL2 - 1].TailPosition := dataHeigh.parameters.Detection.Basic.iSensorPosition + dataHeigh.parameters.Detection.Basic.iMediaFilter;
	END_IF

	AddMediaTrackingEvents(diTotalCmBelt, TAIL_DETECTED, ADR(TrackingEventsArray));

END_ACTION

ACTION CheckExitingMedia:

	//Move out media that hasn't been properly detected
	IF dataHeigh.parameters.Detection.Basic.xEnableMediaTracking THEN
		// If the tail is 50cm far away from the exiting position, move it out
		IF MediaTrackingInsideL1[0].TailPosition > iRejectLengthAdjustment + 50 THEN
			NewMediaExitingL1;
			iForcedMovedOutMediaL1 := iForcedMovedOutMediaL1 + 1;
		END_IF
		// If the tail is 50cm far away from the exiting position, move it out
		IF MediaTrackingInsideL2[0].TailPosition > iRejectLengthAdjustment + 50 THEN
			NewMediaExitingL2;
			iForcedMovedOutMediaL2 := iForcedMovedOutMediaL2 + 1;
		END_IF
	END_IF

	// Run the exact positions moved to avoid detecting the begining of a board more than once
	FOR iIndexExitingMedia := iRejectLengthAdjustment TO iRejectLengthAdjustment + iPositionsToRunArray - 1 DO
		// Detecting the end of a board
		IF NOT xMediaTracking[iIndexExitingMedia].INDEXTRACKING_L1 AND xMediaTracking[iIndexExitingMedia + 1].INDEXTRACKING_L1 THEN
			NewMediaExitingL1;
			EXIT; //The new board has been detected, so not keep on searching for FALSEs
		END_IF
	END_FOR

	// Run the exact positions moved to avoid detecting the begining of a board more than once
	IF NOT dataHeigh.parameters.xDoubleLine THEN
		RETURN;
	END_IF
	FOR iIndexExitingMedia := iRejectLengthAdjustment TO iRejectLengthAdjustment + iPositionsToRunArray -1 DO
		// Detecting the end of a board
		IF NOT xMediaTracking[iIndexExitingMedia].INDEXTRACKING_L2 AND xMediaTracking[iIndexExitingMedia + 1].INDEXTRACKING_L2 THEN
			NewMediaExitingL2;
			EXIT; //The new board has been detected, so not keep on searching for FALSEs
		END_IF
	END_FOR

END_ACTION

ACTION NewMediaExitingL1:

	iBoardsBelowBlockL1 := UINT_SUB(iBoardsBelowBlockL1,1);
	MoveMediaFromInsideToOutL1;

END_ACTION

ACTION NewMediaExitingL2:

	iBoardsBelowBlockL2 := UINT_SUB(iBoardsBelowBlockL2,1);
	MoveMediaFromInsideToOutL2;

END_ACTION

ACTION SensorsArrayAndProductDetectIncoherence:
	//L1
	//Define review range
	IF iProductDetectSensorPosition >= iPositionsToRunArray THEN
		// Not used max because substracting two UINT, instead of negative can be a maximum value
		iFirstIndex := iProductDetectSensorPosition - iPositionsToRunArray;
	ELSE
		iFirstIndex := 0;
	END_IF
	iLastIndex := iProductDetectSensorPosition + dataHeigh.parameters.Detection.ProductDetect.iMediaFilter + iPositionsToRunArray;

	//Review MediaPresentArray
	IF EDGEPOS(xMediaTracking[iProductDetectSensorPosition + dataHeigh.parameters.Detection.ProductDetect.iMediaFilter].INDEXTRACKING_L1) THEN
		xDetectionSystemIncoherenceL1:=TRUE;
		FOR iIndexReviewArray:=iFirstIndex TO iLastIndex DO
			IF xMediaPresentArray[iIndexReviewArray] THEN
				xDetectionSystemIncoherenceL1:=FALSE;
				EXIT;
			END_IF
		END_FOR
	END_IF

	IF NOT (xMediaTracking[iProductDetectSensorPosition].INDEXTRACKING_L1) THEN
		xDetectionSystemIncoherenceL1:=FALSE;
	END_IF

	dataHeigh.status.MediaPosition.L1.xDetectionSystemIncoherence := xDetectionSystemIncoherenceL1;

	//L2
	IF NOT dataHeigh.parameters.xDoubleLine THEN
		RETURN;
	END_IF

	//Define review range
	IF iProductDetectSensorPosition >= iPositionsToRunArray THEN
		// Not used max because substracting two UINT, instead of negative can be a maximum value
		iFirstIndex := iProductDetectSensorPosition - iPositionsToRunArray;
	ELSE
		iFirstIndex := 0;
	END_IF
	iLastIndex := iProductDetectSensorPosition + iPositionsToRunArray;

	//Review MediaPresentArray
	IF EDGEPOS(xMediaTracking[iProductDetectSensorPosition].INDEXTRACKING_L2) THEN
		xDetectionSystemIncoherenceL2:=TRUE;
		FOR iIndexReviewArray:=iFirstIndex TO iLastIndex DO
			IF xMediaPresentArray[iIndexReviewArray] THEN
				xDetectionSystemIncoherenceL2:=FALSE;
				EXIT;
			END_IF
		END_FOR
	END_IF

	IF NOT (xMediaTracking[iProductDetectSensorPosition].INDEXTRACKING_L2) THEN
		xDetectionSystemIncoherenceL2:=FALSE;
	END_IF

	dataHeigh.status.MediaPosition.L2.xDetectionSystemIncoherence := xDetectionSystemIncoherenceL2;

END_ACTION
```

#### PositionArray.st
```iecst
ACTION SubstracDistances:

	(*Less 10 mm to calculate empty belt distance*)
	iDistanceWorkEmptyBelt := UINT_SUB( iDistanceWorkEmptyBelt, iPositionsToRunArray);

	(*Less 10mm to calculate mounted tile out of machine*)
	iDistanceMountPieceOut := UINT_SUB(iDistanceMountPieceOut,iPositionsToRunArray);

	(*Less 10mm to calculate mounted tile out of machine*)
	iDistanceMediaInside := UINT_SUB(iDistanceMediaInside,iPositionsToRunArray);
	iDistanceVirtualMediaInside := UINT_SUB(iDistanceVirtualMediaInside,iPositionsToRunArray);
	iDistanceMediaToRejectInside := UINT_SUB(iDistanceMediaToRejectInside,iPositionsToRunArray);
	iDistanceTrackingEmpty := UINT_SUB(iDistanceTrackingEmpty, iPositionsToRunArray);

	iDistanceBeltTurn := UINT_SUB(iDistanceBeltTurn,iPositionsToRunArray);

	diTotalCmBelt := diTotalCmBelt + iPositionsToRunArray;

END_ACTION

ACTION LoadDistancesBeltRunning:

	// Load Empty belt distance & Media Inside distance
	IF dataHeigh.Inputs.xVirtualMedia THEN
		iDistanceWorkEmptyBelt := dataHeigh.parameters.Belt.iDistanceEmptyBeltIni;
		// Not considering virtual media with Stack enabled
		iDistanceVirtualMediaInside := dataHeigh.parameters.Belt.iDistanceEmptyBeltIni + REAL_TO_UINT(dataHeigh.parameters.ContinuousMedia.MediaData.rLength);
	END_IF
	IF dataHeigh.status.Detection.xFilteredProductDetectMediaL1 OR  dataHeigh.status.Detection.xFilteredProductDetectMediaL2 THEN
		iPositionAdjusted := iProductDetectSensorPosition + dataHeigh.parameters.Detection.ProductDetect.iMediaFilter;
		iDistanceWorkEmptyBelt := MAX(dataHeigh.parameters.Belt.iDistanceEmptyBeltIni - iPositionAdjusted, iDistanceWorkEmptyBelt);
		iDistanceMediaInside := MAX(dataHeigh.parameters.iTotalBlocksLengh - iPositionAdjusted, iDistanceMediaInside);
		iDistanceTrackingEmpty := MAX(iMaxTrackingPosition - iPositionAdjusted, iDistanceTrackingEmpty);
	END_IF
	IF dataHeigh.status.Detection.xFilteredAnalogSensorMedia THEN
		iPositionAdjusted := dataHeigh.parameters.Detection.Analog.iSensorPosition + dataHeigh.parameters.Detection.Analog.iMediaFilter;
		iDistanceWorkEmptyBelt := MAX(dataHeigh.parameters.Belt.iDistanceEmptyBeltIni - iPositionAdjusted, iDistanceWorkEmptyBelt);
		iDistanceMediaInside := MAX(dataHeigh.parameters.iTotalBlocksLengh - iPositionAdjusted, iDistanceMediaInside);
		iDistanceTrackingEmpty := MAX(iMaxTrackingPosition - iPositionAdjusted, iDistanceTrackingEmpty);
	END_IF
	IF dataHeigh.status.Detection.xFilteredArraySensorMedia THEN
		iPositionAdjusted := dataHeigh.parameters.Detection.Array.iSensorPosition + dataHeigh.parameters.Detection.Array.iMediaFilter;
		iDistanceWorkEmptyBelt := MAX(dataHeigh.parameters.Belt.iDistanceEmptyBeltIni - iPositionAdjusted, iDistanceWorkEmptyBelt);
		iDistanceMediaInside := MAX(dataHeigh.parameters.iTotalBlocksLengh - iPositionAdjusted, iDistanceMediaInside);
		iDistanceTrackingEmpty := MAX(iMaxTrackingPosition - iPositionAdjusted, iDistanceTrackingEmpty);
	END_IF
	IF dataHeigh.status.Detection.xFilteredBasicDetectionMedia THEN
		iPositionAdjusted := dataHeigh.parameters.Detection.Basic.iSensorPosition + dataHeigh.parameters.Detection.Basic.iMediaFilter;
		iDistanceWorkEmptyBelt := MAX(dataHeigh.parameters.Belt.iDistanceEmptyBeltIni - iPositionAdjusted, iDistanceWorkEmptyBelt);
		iDistanceMediaInside := MAX(dataHeigh.parameters.iTotalBlocksLengh - iPositionAdjusted, iDistanceMediaInside);
		iDistanceTrackingEmpty := MAX(iMaxTrackingPosition - iPositionAdjusted, iDistanceTrackingEmpty);
	END_IF

	IF dataHeigh.status.Detection.xMediaToRejectDetected THEN
		dataHeigh.Internal.xMediaToRejectTreated := TRUE;
		iDistanceMediaToRejectInside := dataHeigh.parameters.iTotalBlocksLengh;
	END_IF

	//DELOREAN-668
	IF iDistanceBeltTurn = 0 THEN
		dataHeigh.status.Belt.iBeltTurns := dataHeigh.status.Belt.iBeltTurns + 1;
		iDistanceBeltTurn := dataHeigh.parameters.Belt.iBeltPerimeterLength;
	END_IF

END_ACTION

ACTION LoadDistancesAlways:

	//Mounted media evaluation
	IF xMountedMedia THEN
		iDistanceMountPieceOut:= iTotalBlocksLengh;  // Updated iDistanceMountPieceOut to 500;
	END_IF

END_ACTION

ACTION BoardsBelowBlockManagement:

	dataHeigh.status.MediaPosition.iBoardsBelowBlock := 0; //iBoardsBelowBlockL1 + iBoardsBelowBlockL2;  //Just 0 because Sw is not managing properly
	dataHeigh.status.MediaPosition.L1.iBoardsBelowBlock := iBoardsBelowBlockL1;
	dataHeigh.status.MediaPosition.L2.iBoardsBelowBlock := iBoardsBelowBlockL2;

END_ACTION
```

#### ReviewReject.st
```iecst
ACTION FastReviewReject:

	iIndexPositionToReviewMedia:= iRejectLengthAdjustment - MAX(1, iPositionsToRunArray + 2); //Increasing the quantity of data to avoid not checking any position during accelerations

	IF dataHeigh.parameters.Reject.RejectBoardEdge = REJECT_REAR THEN

		//Full stacker requires to set reject order (digital output) when boards "tail" is just about to exit printer's belt
		FOR iIndexMediaPresent := iRejectLengthAdjustment TO iIndexPositionToReviewMedia BY -1 DO
			IF xMediaTracking[iIndexMediaPresent+1] > 0 AND xMediaTracking[iIndexMediaPresent] = 0 THEN
				IF ValidMedia[iIndexMediaPresent] = MEDIATRACKING_INVALID THEN
					xReject:=TRUE;
					//DELOREAN-981: Counting reject orders executed while printing
					dataHeigh.status.Reject.iBoardsRejected := dataHeigh.status.Reject.iBoardsRejected + 1;
					EXIT;
				END_IF
			END_IF
		END_FOR

	ELSIF dataHeigh.parameters.Reject.RejectBoardEdge = REJECT_FRONT THEN

		//Bundle stacker requires to set reject order (digital output) when boards "head" is just about to exit printer's belt
		FOR iIndexMediaPresent := iRejectLengthAdjustment TO iIndexPositionToReviewMedia BY -1 DO
			IF xMediaTracking[iIndexMediaPresent] > 0 AND xMediaTracking[iIndexMediaPresent+1] = 0 THEN
				IF ValidMedia[iIndexMediaPresent] = MEDIATRACKING_INVALID THEN
					xReject:=TRUE;
					//DELOREAN-981: Counting reject orders executed while printing
					dataHeigh.status.Reject.iBoardsRejected := dataHeigh.status.Reject.iBoardsRejected + 1;
					EXIT;
				END_IF
			END_IF
		END_FOR

	END_IF

	//[RGP] We defined during tests with AVT (Zeev and Jordi) that camera gives us the signal whenever we want,
	// so has to be configured with the distance from camera to end of belt.
	//These lines are useful whether Noam camera's reject signals works the same way
	tp_Reject(IN:=(dataHeigh.Commands.xCameraDefectDetected OR xReject), PT:=T#20MS); //Stacker requires a 20ms pulse to active the reject
	tp_RejectLongTime(IN:=((dataHeigh.Commands.xCameraDefectDetected AND dataHeigh.parameters.xBlockInPrint) OR xReject), PT:=T#1500ms); // This variable is to monitorize it more easily
	xReject:=FALSE; //Reset var after using it in the TP

	dataHeigh.Outputs.xReject := tp_Reject.Q;
	dataHeigh.status.Reject.xRejecting := tp_RejectLongTime.Q;

END_ACTION
```

#### Sections.st
```iecst
ACTION LoadSectionsInformation:

	FOR iIndexSection:=1 TO iTotalSections DO
		IF (NOT dataHeigh.status.MediaPosition.xMountedMediaInside) THEN
			//Assign the Max
			dataHeigh.status.Heigh.rMaxHeigh[iIndexSection] := UINT_TO_REAL(iMaxHeigh[iIndexSection])/100;

		ELSIF dataHeigh.Commands.xAllowToSetMountedMediaHeigh THEN
			dataHeigh.status.Heigh.rMaxHeigh[iIndexSection] := dataHeigh.parameters.rMountedMediaHeigh;
		END_IF

		//Increase signal
		//If the condition is OK, raise the signal
		IF iLastMaxHeigh[iIndexSection] < iMaxHeigh[iIndexSection] THEN
			dataHeigh.status.Heigh.xIncreasedHeigh[iIndexSection] := TRUE;
			iCountIncrease[iIndexSection]:=8; //The cycles to have the signal of the increased enabled (to use it in slow programs)
		END_IF
		//Deactivate the signal once the counter arrives
		IF iCountIncrease[iIndexSection]=0 THEN
			dataHeigh.status.Heigh.xIncreasedHeigh[iIndexSection] := FALSE;
		END_IF
		//Reduce the counter related to increase
		IF iCountIncrease[iIndexSection]>0 THEN
			iCountIncrease[iIndexSection] := iCountIncrease[iIndexSection] -1;
		END_IF

		//dataHeigh.status.Heigh.xIncreasedHeigh[iIndexSection] := iLastMaxHeigh[iIndexSection] < iMaxHeigh[iIndexSection];
		iLastMaxHeigh[iIndexSection] := iMaxHeigh[iIndexSection];
	END_FOR

END_ACTION
```
